(* IEC 61131-3 sources: ml2plc/examples/models/structured_text (part 8) *)

(* ---- test5_13k.st ---- *)
FUNCTION_BLOCK NeuralNetworkFB

VAR_INPUT
    input_data : ARRAY[0..4] OF REAL;
END_VAR

VAR_OUTPUT
    output_data : ARRAY[0..2] OF REAL;
END_VAR

VAR CONSTANT
    weights_0 : ARRAY[0..639] OF REAL := [0.087884, 0.019861, -0.120645, 0.107147, 0.108510, -0.209824, 0.028247, -0.067439, -0.017955, -0.147290, -0.044152, 0.074469, -0.058888, 0.021687, 0.118680, 0.075522, 0.073631, 0.110030, -0.236657, -0.068495, 0.032454, -0.131920, 0.026285, 0.065899, 0.005899, -0.086759, -0.068999, 0.126513, 0.120250, -0.038000, -0.006767, 0.065750, -0.029117, -0.015027, -0.120319, -0.212539, -0.105368, 0.074505, -0.034129, -0.051312, 0.169426, -0.112692, -0.026185, -0.089530, -0.065181, 0.010042, -0.051896, 0.010617, 0.083632, 0.159610, 0.026174, -0.171285, 0.004264, -0.070313, -0.094491, -0.141654, -0.152467, -0.156618, 0.092858, 0.118828, -0.052229, 0.008375, 0.033061, -0.192688, 0.001746, -0.046752, -0.129324, 0.150817, 0.004261, -0.119102, 0.039470, 0.110854, 0.036013, 0.111391, 0.032649, -0.101358, 0.029517, 0.081127, -0.131120, 0.030191, -0.073921, -0.066215, -0.138857, 0.117446, -0.204267, -0.076552, -0.113729, -0.110411, -0.046143, -0.050134, -0.177807, -0.017884, -0.068962, 0.016712, 0.066131, -0.097737, -0.106193, 0.097484, 0.054137, 0.121767, 0.109686, 0.092542, 0.089354, -0.074552, -0.203123, 0.140532, 0.141643, 0.060210, 0.020210, -0.161035, -0.144116, 0.140873, 0.103789, 0.073508, 0.004795, -0.115107, 0.086948, -0.059466, 0.117073, 0.013680, -0.031496, -0.164868, -0.113202, -0.082604, -0.006095, -0.168162, -0.110567, 0.046874, 0.136677, -0.073749, -0.155012, 0.014878, -0.081808, 0.120516, 0.058027, 0.145353, -0.058555, 0.169970, 0.055944, -0.106464, -0.128222, 0.048024, -0.034696, 0.045333, -0.081858, -0.044126, 0.116255, -0.032645, 0.032003, -0.076957, -0.143227, -0.022855, 0.031258, -0.128789, -0.003603, -0.048892, -0.177628, -0.061286, -0.205522, -0.115107, 0.037776, -0.058937, 0.105858, -0.171562, -0.111364, 0.005641, 0.013799, -0.030156, -0.012579, 0.138731, 0.152130, -0.132872, 0.006697, 0.030615, 0.032380, 0.099033, -0.036929, -0.106096, 0.088105, 0.045451, -0.001212, -0.054999, 0.011836, -0.200356, 0.118485, -0.131535, -0.076382, -0.113409, -0.136508, -0.098254, -0.114961, -0.107293, 0.082311, 0.142847, 0.215688, -0.091563, -0.096765, 0.206613, -0.199051, -0.171045, 0.031297, 0.036175, -0.169052, 0.002642, 0.031713, -0.080200, 0.119600, -0.076829, 0.080139, 0.087728, 0.077741, -0.114895, 0.089789, 0.080168, 0.076910, -0.097419, 0.053509, -0.025485, 0.138235, -0.007267, -0.163736, 0.012899, 0.039587, -0.003616, -0.071788, -0.133374, 0.202067, 0.095088, -0.135328, 0.047618, -0.138865, 0.097218, -0.084921, -0.171197, -0.132809, -0.030269, -0.199631, 0.071125, 0.096722, -0.117543, 0.109680, 0.125666, -0.187342, 0.017445, -0.181086, -0.113749, -0.160243, 0.146440, 0.145078, -0.233663, -0.124617, 0.020189, 0.104925, 0.091885, 0.136374, -0.015601, -0.137955, 0.067880, 0.188922, -0.114488, 0.006490, -0.073870, 0.020977, -0.157864, 0.083543, 0.024444, -0.012612, -0.184603, -0.155885, 0.037704, 0.041224, -0.191320, -0.026819, -0.137896, -0.026415, 0.037044, -0.009771, 0.196403, 0.007078, -0.052965, 0.021385, 0.019141, 0.128097, 0.099409, -0.082667, -0.044388, -0.141733, 0.008215, 0.058057, -0.006857, -0.162652, 0.131042, -0.070709, 0.116382, -0.018573, -0.097403, -0.185227, 0.072037, -0.193845, 0.027885, -0.064402, -0.099111, -0.093831, 0.008709, 0.068151, -0.170941, -0.121179, 0.017150, -0.059804, -0.133350, 0.123899, 0.176413, -0.016766, 0.089295, 0.127591, -0.040662, -0.062021, 0.035431, 0.069664, 0.023847, -0.041006, -0.117259, -0.124652, -0.044356, -0.079393, -0.063249, 0.124950, 0.164965, -0.199731, 0.063873, 0.134956, -0.238765, 0.055125, -0.055810, 0.051782, 0.056541, 0.108808, -0.073532, -0.077848, 0.123551, 0.024601, -0.120728, -0.004044, 0.112966, -0.161989, 0.012075, -0.070966, -0.124047, 0.167929, 0.125195, 0.098143, -0.096104, 0.166867, 0.114795, -0.136621, -0.019339, 0.168998, -0.007273, 0.138194, 0.038277, 0.112113, -0.097517, 0.167485, 0.052191, -0.080308, 0.085419, 0.078983, -0.111131, -0.060336, -0.188764, 0.007864, 0.047479, -0.094697, 0.132104, -0.231222, -0.136076, 0.007164, 0.140243, 0.200802, -0.160538, 0.028893, 0.105251, -0.087435, -0.023133, -0.181240, 0.031476, -0.069354, 0.025107, 0.003484, 0.017893, 0.013283, 0.086928, 0.116381, -0.105047, -0.011669, -0.144326, -0.081993, 0.015335, 0.162402, 0.170721, -0.073380, -0.064310, 0.021418, -0.052916, -0.194195, -0.104925, 0.077744, -0.046308, 0.041450, 0.123528, -0.009889, 0.048534, -0.204614, 0.114375, -0.007900, -0.096067, -0.144443, 0.066950, -0.017162, 0.127650, -0.021940, -0.186933, -0.174070, 0.114869, 0.013821, 0.049158, 0.118836, 0.110080, -0.179380, -0.145327, -0.151734, -0.067201, 0.090523, -0.180013, -0.111317, 0.028459, 0.011573, 0.167342, 0.032929, -0.037529, 0.162289, 0.121033, 0.033484, 0.080197, -0.115669, -0.150395, 0.122810, -0.140164, 0.012817, -0.085399, -0.030360, 0.052412, 0.199205, -0.085308, 0.099355, -0.185208, -0.119913, 0.022915, -0.003856, 0.096522, -0.164929, -0.085813, -0.083492, 0.066105, -0.127158, 0.160928, 0.150646, -0.064350, -0.094705, 0.068810, 0.104658, 0.100290, 0.016024, 0.107678, 0.176333, 0.074564, -0.097281, -0.158018, -0.189581, -0.098518, -0.040255, -0.200370, -0.032509, -0.113215, -0.046972, -0.175030, 0.121636, 0.006522, 0.068477, 0.060772, -0.172631, 0.022521, -0.104405, -0.176789, 0.053084, -0.234425, -0.225009, 0.077532, 0.060609, -0.072898, -0.043883, -0.159845, 0.054400, -0.060357, 0.152364, 0.075698, -0.101363, 0.156116, -0.068740, -0.008421, 0.115683, -0.032726, 0.049882, 0.060400, -0.041212, -0.130228, 0.171733, -0.081668, -0.138404, 0.156815, -0.057446, 0.156922, 0.138291, 0.004256, 0.156900, -0.256590, -0.045184, 0.056040, 0.093967, -0.093704, 0.088963, -0.071382, 0.138222, 0.082414, 0.019420, 0.140588, -0.114552, -0.081097, -0.043554, -0.027499, -0.167955, 0.141868, 0.030455, 0.116915, 0.078890, -0.036069, -0.054053, 0.126143, 0.016059, 0.096736, 0.161875, 0.148323, -0.004357, -0.166265, -0.138691, 0.038991, 0.137727, 0.012094, -0.163153, -0.058560, -0.009588, -0.142637, -0.131980, 0.059672, -0.001274, -0.182290, -0.218865, -0.117359, -0.147914, 0.161844, -0.171897, -0.093763, 0.165442, 0.016261, -0.184435, -0.071222, 0.075867, -0.019360, -0.157325, -0.025250, -0.191039, 0.152266, -0.070228, -0.082297, 0.103244, -0.262244, 0.154374, 0.147566, -0.188977, -0.058970, 0.071598, 0.084986, -0.117181, -0.221621, -0.140587, -0.165058, 0.133049, -0.004266, -0.108147, 0.034074, -0.004569, -0.023090, 0.005967, -0.013832, -0.056172, 0.101765, -0.228049, 0.212225, -0.149336, -0.038122, -0.155115, 0.051004, -0.012800, 0.093140, -0.253202, -0.082567, -0.049787, 0.180747, -0.041803, 0.003407, 0.064646, 0.024799, -0.096398, 0.025533, -0.177775, -0.043537, -0.056790, -0.013036, -0.173823, 0.109881, 0.120896, 0.023794, -0.107422, -0.086024, 0.180928, -0.020671, 0.083740, 0.123611, 0.087525, 0.156801];
    bias_0 : ARRAY[0..127] OF REAL := [-0.138056, -0.724342, -0.149341, -0.281606, -0.725367, 0.232611, -0.248216, -0.224301, -0.455382, -0.588808, 0.331585, -0.105728, -0.004159, 0.141275, -0.052369, -0.498210, -0.228472, 0.128578, -0.324100, -0.114577, -0.552493, -0.092725, -0.231976, -0.594564, 1.152468, 0.320418, 1.080323, -0.436585, -0.201718, -0.644658, -0.083568, 0.892163, -0.533870, 0.395853, 0.012269, 0.399186, -0.090490, -0.443884, 0.422784, 0.699066, 0.525596, -0.248559, 0.707993, 0.283335, 0.051301, 0.005778, 0.071785, 0.709974, -0.306237, 0.124496, 0.201839, -0.570137, -0.169047, -0.182123, 0.495954, -0.100448, 1.026744, -0.484968, 0.789213, 0.337440, 0.164353, -0.134713, -0.277190, 0.014476, -0.957523, -0.088268, 0.004471, -0.558361, 0.308556, -0.375165, -0.692890, 0.276062, 0.256898, 0.133769, -0.481402, -0.289402, -0.027431, 0.037170, 0.774907, -0.558535, -0.040130, 0.377911, 0.574793, 0.486151, 0.168924, 0.406046, 0.144867, -0.593385, 0.075902, -0.426114, -0.372866, 0.453651, -0.236809, -0.562530, 0.037890, -0.083074, -0.047217, 0.078249, 0.167289, -0.330759, -0.283430, -0.460562, -0.174557, 0.892016, -0.115629, -0.579056, 0.747610, -0.564211, -0.082146, 0.059292, 0.430699, 0.005029, 0.198333, -0.513879, 0.096918, 0.126206, 0.071723, -0.133315, -0.245988, 0.964687, -0.703479, 0.089156, -0.414976, -0.108005, -0.900232, -0.744488, -0.873102, -0.797852];

    weights_1 : ARRAY[0..12287] OF REAL := [-0.081575, -0.080771, 0.015952, -0.039088, -0.116122, 0.043837, 0.081503, -0.146702, -0.097420, 0.123321, -0.143534, 0.087642, -0.013072, 0.120403, -0.032723, -0.019567, 0.109142, 0.046921, -0.151230, 0.034047, 0.068958, -0.110997, -0.006236, 0.099731, 0.103434, -0.019739, 0.061900, -0.030395, -0.006606, 0.042065, 0.125518, -0.158020, -0.060671, -0.011133, -0.174419, -0.000909, -0.087395, 0.107763, 0.032645, -0.159583, 0.019297, -0.055804, 0.041226, -0.102607, 0.111457, 0.036441, 0.020504, 0.026678, 0.022357, 0.058828, 0.009128, -0.137546, 0.099089, -0.132678, -0.139020, -0.078414, 0.134850, -0.109238, -0.088241, 0.086606, -0.129975, -0.106856, -0.173047, 0.002129, 0.073779, -0.001719, 0.012466, -0.149798, 0.068260, 0.018230, -0.073247, 0.025459, -0.025935, -0.083550, -0.014844, 0.044535, 0.024790, 0.031258, 0.047537, -0.126853, 0.030907, -0.174494, 0.123196, -0.139801, -0.101418, -0.042713, -0.031737, -0.139095, -0.141767, 0.051548, -0.103749, -0.134006, 0.124273, 0.033699, 0.088179, -0.196681, -0.061558, -0.097976, 0.041162, -0.066488, -0.223767, -0.156958, 0.119515, 0.030284, 0.064781, 0.065118, -0.019679, -0.014793, 0.070956, 0.005814, -0.125978, 0.148016, -0.176253, -0.110496, -0.086278, -0.064303, 0.029931, 0.013686, 0.164138, -0.022327, -0.030191, 0.187196, -0.098539, -0.023848, 0.048127, -0.111411, -0.095664, -0.256552, 0.008552, -0.103314, 0.051327, -0.022576, -0.091046, 0.019166, -0.099166, -0.173986, -0.026153, 0.027388, -0.109343, 0.046421, 0.037128, -0.124205, -0.198771, 0.073731, -0.039520, 0.016815, -0.047930, -0.129724, 0.019335, -0.119635, -0.026225, -0.029072, 0.158678, -0.173663, 0.027847, -0.049243, -0.020055, -0.109040, 0.095462, -0.042686, 0.151513, -0.077091, -0.131769, 0.054254, 0.026624, -0.155398, -0.082870, -0.159275, 0.059890, 0.062534, -0.142575, -0.059085, -0.185808, -0.137954, -0.029401, 0.077038, 0.112156, 0.029459, 0.065796, 0.013224, -0.179952, -0.117919, -0.115410, 0.092213, 0.008067, 0.144769, -0.132419, 0.141382, -0.085988, -0.073259, -0.108810, -0.089521, 0.090714, 0.070094, 0.051771, -0.198376, 0.097630, 0.134390, 0.070879, -0.084352, -0.077932, -0.084724, 0.013531, 0.103697, 0.083068, -0.022807, -0.099833, 0.026875, -0.011101, 0.100574, -0.189504, 0.008358, -0.130581, -0.017598, 0.049774, -0.038556, -0.034455, 0.092771, 0.008732, -0.099842, -0.203902, 0.097001, 0.054298, 0.068758, -0.017547, -0.119806, -0.001483, 0.150792, 0.059175, -0.024380, 0.077527, -0.089932, -0.095934, 0.067083, 0.051638, -0.140169, 0.016767, -0.031886, -0.077586, -0.156478, 0.136940, -0.068401, -0.156731, -0.031153, 0.027569, -0.069691, 0.016632, 0.085590, -0.087230, -0.124976, 0.178376, 0.054593, 0.139863, 0.138583, -0.028121, -0.011154, -0.060567, -0.100126, -0.094427, -0.078613, -0.021682, -0.123174, -0.107229, 0.095945, -0.081012, -0.122688, -0.075887, -0.142662, -0.036621, -0.064916, -0.071555, 0.096564, 0.021082, 0.004940, 0.073835, 0.102978, 0.013753, -0.087000, -0.023456, -0.025726, 0.041069, 0.019725, -0.170109, -0.065330, -0.065098, -0.043905, -0.013389, -0.033329, 0.077615, 0.045581, -0.113043, -0.026083, -0.092637, 0.131571, 0.111947, 0.053334, 0.064196, -0.046716, -0.096859, -0.185973, -0.034940, 0.044770, -0.124819, 0.029667, -0.082584, -0.149761, -0.067224, 0.100945, 0.101797, -0.123318, 0.079437, -0.170388, 0.043855, -0.096770, 0.093361, -0.037078, -0.054357, -0.136876, 0.030271, 0.088059, -0.158535, 0.016276, -0.199991, -0.136451, -0.101051, -0.099338, -0.051318, -0.091107, -0.092926, 0.125917, 0.120004, 0.099235, 0.054448, -0.054184, -0.088516, 0.031720, -0.110417, 0.021548, 0.114272, 0.104105, -0.029168, -0.104910, 0.043389, 0.110131, 0.067098, 0.063883, 0.125061, -0.140973, -0.087429, -0.183545, 0.001501, 0.090085, 0.090463, -0.068449, 0.104290, -0.047815, -0.107690, 0.142746, -0.009204, -0.074146, 0.109043, -0.056259, 0.005365, -0.095835, -0.019732, -0.090880, -0.179324, -0.144838, 0.008955, -0.031656, -0.153258, -0.049975, -0.136535, -0.153729, -0.007882, 0.076208, -0.147986, 0.120409, -0.050599, 0.102071, 0.002109, -0.156943, -0.029278, -0.102693, -0.051444, 0.111964, 0.059902, -0.168826, -0.068986, -0.174917, 0.080254, 0.004751, 0.066618, 0.096905, 0.066631, -0.175463, 0.091283, -0.263883, 0.056194, 0.079930, -0.117990, -0.009883, 0.138474, -0.146369, -0.138613, -0.192223, -0.044161, 0.087972, 0.023354, 0.044543, 0.110326, -0.011888, 0.100713, 0.032271, -0.142762, -0.173276, -0.082045, -0.071345, -0.156709, -0.059416, 0.024078, 0.016129, 0.006350, -0.202165, -0.177114, 0.204796, 0.039982, -0.145523, 0.047530, -0.165438, 0.029745, -0.033077, 0.192667, -0.125515, -0.130639, 0.063787, -0.023226, 0.007809, -0.015500, 0.005910, 0.012534, -0.158731, -0.177921, -0.028937, -0.156686, -0.188195, 0.135282, 0.209456, 0.003387, -0.116251, -0.139349, 0.030706, 0.084070, 0.139131, -0.130020, 0.098266, -0.017343, -0.102753, -0.081793, -0.108168, 0.015434, -0.063223, -0.088817, 0.008182, 0.044385, 0.194167, 0.068721, 0.144784, -0.144739, 0.149692, -0.122958, 0.034189, -0.118378, -0.035300, -0.031611, -0.090980, 0.098072, -0.082291, 0.040535, 0.028408, 0.077057, 0.016835, -0.177612, -0.111623, 0.112017, -0.175378, 0.122941, 0.071300, -0.029213, -0.042673, -0.095251, 0.091868, -0.124875, 0.123380, 0.094310, -0.056404, 0.101097, -0.187158, -0.099725, -0.074531, -0.119461, -0.089910, 0.027321, -0.089037, -0.095327, -0.095788, 0.158980, -0.080355, 0.051269, -0.036277, 0.013874, 0.087641, 0.023480, -0.123195, -0.114087, 0.079653, -0.005070, 0.083194, 0.071204, -0.012910, -0.128791, -0.214303, 0.041115, -0.126938, 0.010794, -0.104911, -0.167860, -0.056907, 0.149767, 0.072014, 0.018457, -0.003708, -0.084242, 0.034660, 0.148553, 0.060466, 0.050078, 0.173174, -0.156669, 0.012732, -0.156297, -0.083725, -0.087539, -0.276414, -0.029359, -0.057753, 0.001603, 0.126020, -0.011550, 0.082022, -0.048681, -0.161668, 0.021370, 0.141360, -0.130907, -0.191119, -0.010477, -0.036678, -0.091980, 0.101416, -0.012654, -0.061183, -0.145007, 0.024690, 0.037292, 0.001704, 0.096528, -0.209641, 0.002475, -0.044156, -0.063900, 0.157965, -0.209313, 0.107978, -0.030685, 0.127991, 0.088548, -0.137926, -0.008005, -0.103959, 0.038476, 0.099615, -0.041820, 0.010803, -0.100065, 0.066539, -0.149380, 0.131097, -0.141308, -0.049057, -0.054971, -0.036114, 0.115146, -0.148750, -0.126427, -0.078635, -0.048640, -0.046237, -0.130117, 0.004752, 0.102776, -0.069640, 0.024115, -0.109310, -0.096013, 0.116772, -0.136342, -0.151241, -0.199084, 0.039571, 0.116098, -0.054730, -0.043315, 0.050230, 0.093377, -0.058800, 0.043897, -0.096458, 0.167670, -0.171068, 0.003364, -0.012613, 0.132328, 0.043677, 0.004500, -0.052957, -0.181461, 0.092122, 0.161901, -0.018877, 0.097804, -0.101418, 0.057685, 0.046452, 0.063500, -0.149884, -0.077202, -0.050282, 0.062265, -0.133137, 0.094386, -0.027847, 0.003860, -0.058797, 0.096755, 0.133752, 0.018234, 0.115755, -0.137680, 0.030889, -0.043614, 0.082428, 0.045449, 0.049964, 0.031676, -0.006952, -0.006175, -0.060989, 0.016020, -0.001273, -0.129249, -0.027272, -0.145721, 0.129620, 0.032681, -0.020259, 0.089839, -0.076454, 0.031277, -0.137930, -0.190245, -0.092762, -0.169273, -0.125275, 0.042772, -0.150519, -0.108547, -0.041230, -0.111160, -0.003413, -0.131887, 0.051243, -0.094373, 0.115747, 0.035868, -0.115496, -0.008602, -0.121400, -0.088105, 0.047530, 0.094965, -0.057794, 0.045937, 0.047745, -0.151089, 0.135993, 0.068231, -0.079802, -0.143148, -0.122689, 0.037814, -0.170841, 0.047921, -0.078489, -0.068901, -0.145030, -0.124568, 0.037971, -0.112618, 0.090066, 0.053041, -0.113300, 0.042961, 0.100212, -0.056396, -0.114706, -0.163505, -0.130223, -0.165611, -0.038295, 0.013722, -0.089551, -0.117751, -0.038264, 0.169660, -0.045797, -0.036698, -0.141689, -0.065967, -0.000077, 0.019098, -0.069963, -0.092839, -0.101812, -0.004868, -0.023554, -0.133523, -0.142896, 0.034829, 0.025655, 0.172733, -0.116783, 0.116567, 0.077891, 0.170584, 0.107316, -0.126802, -0.021477, -0.087033, 0.107559, -0.062535, 0.110244, -0.020078, 0.006528, -0.196714, -0.008804, -0.034624, -0.037185, -0.040095, -0.127234, -0.015266, -0.029318, 0.098768, 0.070560, -0.188236, 0.091512, 0.072778, -0.121254, -0.142115, -0.102058, -0.126129, -0.144473, 0.047309, 0.031633, 0.111848, 0.022209, 0.000316, -0.103872, -0.152406, 0.063265, -0.086201, -0.049895, -0.128511, -0.042608, -0.013025, 0.129606, -0.152738, 0.091822, -0.170736, -0.122971, 0.036491, -0.103669, -0.093657, 0.065951, 0.086443, -0.007772, 0.126724, 0.061812, 0.073030, -0.227505, -0.150730, -0.152455, 0.003632, -0.019424, -0.054101, 0.081972, 0.112612, 0.019746, 0.076702, 0.212985, -0.150149, -0.038424, -0.126008, 0.020174, -0.003787, -0.029846, 0.013167, 0.071178, -0.081888, 0.097691, 0.020292, 0.018873, -0.140535, 0.051663, -0.155505, 0.038109, -0.005970, 0.018861, 0.061807, 0.091283, 0.099963, 0.122483, 0.048785, 0.033977, 0.041410, 0.140400, -0.092338, 0.112759, 0.076005, -0.133343, -0.162613, -0.008164, -0.002846, 0.120728, -0.049317, 0.054437, -0.127069, 0.042041, -0.035214, 0.139597, 0.073649, -0.101931, -0.016045, 0.181245, -0.043369, 0.026610, -0.137698, 0.167959, 0.122667, -0.008332, 0.021051, 0.040108, -0.156969, -0.068006, 0.137933, 0.012884, -0.106799, -0.009552, -0.219680, -0.027378, 0.057219, -0.206282, 0.012929, -0.139442, 0.068162, -0.159516, 0.096407, -0.083495, -0.205347, 0.011081, 0.048977, -0.011546, 0.089416, -0.219959, -0.146311, 0.047244, 0.006085, 0.036988, 0.133529, 0.083324, -0.074794, -0.099529, -0.002222, -0.047307, -0.030684, -0.177784, -0.093368, -0.141561, 0.078858, 0.135456, -0.166646, 0.034251, -0.020081, 0.068057, -0.141532, 0.075862, 0.065621, -0.052889, -0.186487, 0.010214, -0.061436, -0.028441, 0.125152, -0.036969, 0.058498, 0.044020, 0.165813, -0.125980, -0.033366, -0.174131, -0.125943, 0.055094, -0.088112, 0.035833, 0.041747, 0.076717, 0.076765, -0.016334, -0.119987, -0.135628, 0.015400, 0.005722, 0.006286, -0.129062, -0.029350, -0.044798, 0.037943, 0.126117, -0.132406, 0.036613, -0.112067, -0.031121, 0.100631, -0.012509, 0.072480, 0.034916, -0.040505, 0.007290, 0.049140, 0.149019, -0.092554, -0.042404, 0.068616, 0.132734, 0.003138, 0.170876, -0.031358, -0.155839, -0.081269, 0.042707, -0.034900, 0.220723, -0.018079, 0.113232, -0.039536, -0.035911, 0.146646, 0.089903, 0.006342, -0.012555, 0.067873, -0.115261, 0.082812, 0.164852, 0.084914, 0.086952, -0.101140, 0.065694, 0.004201, 0.021580, -0.042629, 0.105508, -0.085644, 0.183658, 0.178939, 0.059744, -0.124989, -0.095250, -0.118859, 0.001045, -0.026453, 0.015741, -0.001020, -0.147134, 0.057491, 0.033330, 0.098456, 0.085774, -0.069800, 0.053079, 0.116645, 0.082423, -0.088994, 0.040234, -0.084737, -0.119974, -0.002935, -0.071704, 0.159501, 0.157314, -0.116031, -0.094580, 0.004709, -0.090457, 0.034409, -0.098700, -0.012167, 0.037498, -0.034314, 0.049258, 0.043418, -0.047919, -0.128354, -0.004897, -0.122908, 0.149899, 0.089695, 0.137241, -0.001262, 0.026590, 0.062069, -0.022439, 0.013561, 0.108820, -0.134295, 0.137737, -0.104128, 0.029637, 0.102498, 0.075547, 0.098281, 0.107930, -0.099356, -0.012938, -0.020183, -0.223851, 0.043924, 0.107465, 0.156199, -0.088132, 0.188467, 0.102066, 0.064692, -0.090133, -0.001347, -0.082854, 0.183009, -0.038977, -0.159207, 0.057301, -0.136873, 0.048873, 0.031771, -0.171822, 0.033120, 0.105704, -0.084895, 0.095055, 0.137444, -0.163820, 0.112387, 0.051031, -0.072802, -0.100967, 0.013958, 0.075336, -0.143393, -0.055055, -0.117185, 0.108107, 0.162765, -0.049701, -0.010500, -0.129675, 0.059109, -0.169230, 0.061079, -0.012083, -0.151733, 0.007924, -0.064643, -0.044676, -0.096629, -0.106404, 0.128860, -0.123374, 0.097159, 0.044151, -0.102661, -0.142225, -0.094126, -0.005144, -0.182815, 0.042802, -0.011589, -0.081280, -0.168038, 0.082915, -0.112574, -0.051578, -0.001187, -0.026704, -0.091962, -0.026611, -0.171998, -0.021113, 0.140911, -0.098982, 0.098242, 0.080007, 0.037016, -0.078325, 0.135061, 0.078783, -0.140612, 0.098578, -0.096234, 0.081160, -0.122356, -0.113938, -0.164598, 0.011331, -0.139634, -0.015426, 0.157431, -0.172702, 0.099078, -0.018352, 0.028085, -0.102126, 0.009692, -0.057786, -0.068308, 0.046532, 0.022939, 0.047090, 0.057643, 0.101340, 0.031700, -0.155278, 0.025313, -0.162245, 0.062350, 0.080738, 0.009415, -0.026625, 0.119341, -0.115887, 0.043791, 0.043181, 0.113826, -0.121817, 0.102165, -0.069487, 0.006380, 0.074927, 0.043731, 0.147266, 0.039980, -0.006088, -0.082346, -0.193183, -0.022871, -0.117219, 0.016636, -0.028051, -0.106046, -0.005760, 0.153666, -0.068575, 0.080032, 0.041547, -0.070853, -0.039723, -0.133037, 0.124683, -0.105086, -0.130024, -0.122982, -0.097882, -0.166385, 0.096523, -0.060713, 0.046434, -0.158093, 0.057526, 0.090288, 0.091276, 0.087174, -0.018942, -0.022930, 0.028879, 0.081154, 0.050385, -0.228233, 0.075629, -0.141450, 0.016981, -0.003183, -0.011411, -0.034834, 0.062535, -0.140759, -0.069517, -0.054256, -0.126463, 0.062169, -0.071767, 0.063638, 0.035320, 0.025509, -0.102183, -0.013740, -0.105443, 0.067947, -0.093319, 0.066332, 0.001127, -0.230074, -0.032940, -0.024680, -0.075319, 0.104570, -0.063355, 0.042160, -0.083321, 0.096235, -0.054556, 0.046468, -0.142220, -0.152431, -0.080084, -0.034122, -0.039364, 0.021040, -0.121876, -0.047387, -0.016643, -0.075452, 0.011071, -0.096630, 0.167191, -0.022463, -0.161584, -0.114355, -0.013775, -0.212787, 0.114291, 0.148954, -0.270307, -0.044340, -0.038644, -0.130380, 0.008371, 0.179310, 0.028057, -0.112501, 0.099296, -0.023552, 0.042440, -0.223643, -0.089552, 0.121801, -0.101898, 0.101719, -0.019475, -0.138102, 0.007500, 0.114520, -0.020841, 0.078318, -0.146791, -0.159486, -0.033819, -0.108025, 0.019645, -0.240050, -0.094725, 0.001863, -0.061960, 0.070538, 0.037391, -0.004894, -0.129432, -0.039346, -0.016018, 0.048675, 0.183405, -0.061341, 0.044579, -0.075781, -0.090313, -0.061431, -0.242545, 0.149409, 0.192036, 0.042303, -0.174307, -0.174971, 0.118598, -0.012059, 0.008028, -0.051703, 0.072126, 0.039219, -0.051813, -0.157609, -0.053761, 0.077431, -0.167700, -0.136599, -0.126247, -0.083612, 0.061878, -0.069953, 0.017028, -0.059142, -0.105931, 0.065761, -0.230763, 0.098776, -0.233016, 0.107031, -0.091945, -0.140657, 0.106068, -0.168658, 0.117609, -0.162881, -0.062493, -0.031648, -0.215897, -0.011096, -0.223865, -0.194450, 0.018461, -0.098600, 0.019417, -0.010198, 0.121387, -0.085882, 0.033285, 0.064565, -0.101164, -0.154355, -0.008463, -0.022031, 0.086821, 0.073677, -0.047492, -0.006241, -0.083720, -0.064338, -0.030201, 0.068820, -0.012762, 0.006955, -0.069824, 0.048148, -0.098935, -0.074085, -0.131027, -0.048977, -0.079691, 0.061712, -0.017702, 0.047844, -0.149083, -0.174584, -0.017555, -0.069080, 0.057426, 0.023185, 0.094438, 0.055650, -0.178939, 0.114310, -0.196780, -0.032571, -0.060820, -0.076543, 0.022690, 0.098297, -0.095817, 0.016638, 0.011793, -0.101782, 0.005777, -0.149359, 0.027835, -0.077289, 0.092431, -0.093891, 0.010222, 0.012915, -0.102511, -0.031433, -0.139489, -0.131653, -0.133860, -0.170684, 0.000861, 0.176236, 0.023889, -0.122425, 0.031023, -0.042648, -0.200706, -0.007618, -0.172353, -0.060969, -0.111408, 0.035170, 0.026013, -0.059565, 0.163137, 0.100273, 0.142385, 0.054498, -0.210962, 0.083249, -0.172852, 0.049680, 0.061989, 0.080453, 0.054906, 0.060045, -0.137977, -0.005662, 0.011224, 0.083500, 0.057573, -0.103310, 0.014571, 0.012037, -0.127015, -0.040393, -0.106786, -0.132445, -0.089465, 0.053720, -0.111644, -0.152595, -0.072208, -0.170288, 0.040783, -0.051353, -0.123556, -0.059620, -0.006337, 0.053879, 0.018863, 0.178810, -0.048635, 0.011481, 0.031570, 0.134769, -0.086727, 0.057939, -0.112196, -0.124786, -0.037214, -0.183068, 0.051824, 0.088464, 0.170947, -0.089516, -0.101557, -0.023134, 0.039533, -0.137372, -0.068921, 0.120034, -0.064358, -0.211081, 0.050003, 0.097631, -0.164230, -0.003052, -0.045674, 0.033500, -0.155961, 0.149210, -0.005820, -0.095616, -0.008706, -0.073449, -0.007479, -0.065913, 0.011839, 0.061956, -0.159078, -0.007190, 0.028311, -0.068458, -0.032719, -0.096845, 0.000351, 0.083672, -0.176350, -0.101202, -0.156637, 0.120088, -0.090894, 0.074344, -0.097555, -0.069346, -0.097220, 0.005215, -0.199269, -0.075000, -0.012239, -0.153847, -0.132105, -0.173554, -0.022580, -0.075864, 0.072241, -0.179801, 0.114656, 0.058945, 0.032403, -0.035467, -0.073135, -0.026923, -0.004199, 0.126423, -0.123071, 0.024513, 0.119495, -0.079067, 0.107798, -0.002691, -0.177214, -0.080168, 0.087260, 0.083324, -0.036822, 0.012710, 0.006805, 0.025345, 0.014063, 0.139339, 0.068182, -0.163975, -0.018243, -0.111255, 0.011790, 0.047546, 0.092633, 0.049318, 0.003007, -0.145426, 0.051505, 0.019591, 0.038348, 0.106809, 0.146770, -0.137394, 0.023419, -0.104374, 0.015242, -0.077740, -0.014287, 0.107080, 0.149179, -0.032868, 0.014391, 0.112384, -0.140490, 0.000523, 0.038513, 0.085826, 0.033327, 0.122935, 0.068390, 0.046117, 0.030794, -0.186023, -0.078125, -0.018852, 0.109274, 0.066455, 0.017141, -0.133333, -0.193708, -0.146445, -0.015501, 0.026529, 0.082395, 0.149612, -0.070591, -0.016908, -0.059412, 0.034737, -0.125785, -0.132630, 0.051595, -0.068432, 0.058917, -0.063994, -0.020062, -0.155251, -0.130603, -0.102926, -0.068344, 0.223298, 0.114052, 0.093608, -0.056596, 0.014436, 0.056514, 0.053748, 0.041788, -0.013315, -0.054554, -0.021707, -0.017912, -0.076426, -0.065880, -0.060482, 0.059109, 0.033523, -0.065950, 0.130728, 0.155523, -0.122129, 0.097537, -0.222720, -0.033999, -0.179547, 0.132113, -0.132758, -0.163402, -0.097568, 0.081810, -0.063774, -0.237891, -0.098302, 0.001285, -0.002167, -0.148563, -0.078971, -0.102606, -0.169557, -0.090034, 0.104811, 0.052321, 0.137128, 0.028810, -0.102812, 0.046596, 0.095611, -0.091704, -0.122140, -0.040893, 0.128003, -0.118820, 0.079260, -0.053132, 0.120491, 0.065923, 0.101679, -0.118584, -0.076018, 0.031019, -0.158750, 0.066865, 0.156857, 0.124133, 0.072551, 0.136147, -0.068172, -0.190488, -0.019130, 0.084109, -0.069187, 0.136179, -0.005778, 0.083175, 0.004151, -0.108535, 0.124859, -0.054482, -0.019212, -0.051216, 0.151764, -0.133774, 0.026327, -0.140163, -0.237679, -0.014108, 0.064628, 0.025393, -0.200114, -0.067511, -0.001822, -0.160585, -0.037121, -0.149930, 0.102790, -0.021203, -0.122963, -0.091361, 0.006626, -0.123720, 0.008464, 0.025206, -0.143426, 0.050645, -0.066107, -0.114658, 0.021127, -0.077297, 0.020617, -0.055209, -0.196839, 0.019999, -0.047371, 0.108169, -0.014506, -0.082857, 0.090321, -0.072653, 0.029153, -0.007638, 0.054287, -0.066536, 0.103992, -0.068357, 0.043941, -0.139107, -0.132066, 0.079844, 0.038007, -0.042187, -0.056770, 0.086439, 0.099471, 0.056606, -0.120636, 0.073782, 0.127915, -0.159352, 0.139489, -0.109178, -0.001992, -0.091596, -0.132664, -0.016212, 0.041536, 0.108049, 0.085386, 0.068069, -0.030001, -0.029575, -0.137504, 0.113700, 0.117755, 0.133271, -0.015861, -0.094789, -0.130660, -0.131559, -0.135082, -0.177463, -0.057344, 0.001805, 0.136894, -0.146070, -0.103945, -0.151248, 0.062254, -0.020492, -0.017738, 0.082921, 0.042381, -0.109089, -0.128478, 0.002673, -0.000820, 0.111654, 0.098417, 0.104491, -0.044083, 0.144458, 0.042958, -0.115993, -0.112584, -0.192943, 0.022451, 0.017492, -0.054143, 0.040774, 0.133315, -0.069498, -0.079107, -0.064530, 0.116959, 0.105073, -0.058618, 0.066981, 0.110520, -0.144423, 0.052642, 0.093975, -0.149870, -0.052229, -0.001838, 0.011842, -0.085902, 0.147386, -0.059832, -0.049631, -0.042176, -0.175652, -0.072840, -0.031563, -0.112192, 0.084438, -0.114146, -0.094277, -0.112050, 0.000733, -0.171038, -0.045380, -0.079449, 0.126015, -0.108049, -0.208123, -0.046716, -0.193074, -0.061850, -0.156245, 0.102635, 0.133027, 0.053019, 0.095702, -0.069115, 0.134063, 0.129244, -0.039284, 0.024840, -0.002832, 0.003597, -0.088943, 0.082234, 0.073630, 0.102140, -0.006331, 0.014311, 0.078271, -0.088671, 0.122475, -0.099081, -0.042141, 0.071669, 0.087143, 0.093409, 0.028684, -0.099658, -0.022964, -0.073099, 0.074543, -0.151403, 0.114005, 0.093944, -0.021708, 0.104447, -0.085412, 0.053264, 0.121513, -0.109735, -0.168127, 0.097666, 0.119226, -0.030115, -0.049430, 0.060198, -0.012868, -0.016367, -0.138113, -0.145767, -0.009954, 0.013421, -0.126789, 0.056323, 0.116540, 0.010144, 0.100273, -0.079003, 0.124674, 0.142510, 0.035960, -0.160469, -0.118609, -0.177625, -0.066986, 0.061048, -0.183329, -0.144361, -0.094739, -0.051829, -0.079642, -0.107499, -0.153177, 0.129971, -0.110818, 0.028459, -0.109879, 0.093607, -0.010001, -0.146904, -0.124400, 0.069906, -0.151181, -0.136660, -0.132783, -0.029697, -0.035066, 0.066000, -0.000677, 0.103650, -0.037971, 0.019022, -0.057398, -0.089334, -0.149536, 0.098794, 0.086038, 0.018742, -0.149346, -0.059685, 0.100798, -0.072522, -0.016912, -0.024436, -0.013465, 0.146220, 0.026841, 0.122860, -0.184557, -0.000641, -0.171788, 0.037912, -0.007957, -0.029495, 0.072551, 0.019778, -0.033822, 0.017165, -0.074381, -0.010408, -0.108626, -0.107838, -0.161565, -0.167354, 0.053410, 0.083216, 0.061002, 0.002115, 0.069332, 0.127145, -0.065106, -0.074354, -0.123912, 0.031066, 0.006686, -0.089992, -0.149129, -0.119466, -0.104320, 0.050860, -0.143835, 0.147742, -0.002157, 0.074529, 0.178429, -0.044086, -0.104907, -0.089663, -0.042856, 0.104700, -0.088354, 0.031053, -0.100033, -0.032134, 0.149250, -0.038932, -0.014376, -0.021739, -0.093341, -0.054363, 0.108898, 0.114017, -0.086645, 0.083144, 0.090645, 0.098105, -0.022636, -0.052745, -0.018285, -0.041028, 0.034169, -0.079790, 0.115126, -0.123778, -0.065468, -0.003593, -0.107618, -0.035261, 0.040267, 0.132502, -0.022881, -0.037396, 0.036865, 0.099346, 0.039147, 0.115031, 0.120937, 0.047241, -0.046646, -0.107199, -0.020799, 0.046719, 0.079567, -0.011353, -0.114912, -0.075716, 0.116529, 0.170175, -0.155336, 0.015451, 0.102393, 0.019118, 0.028938, -0.028650, 0.025321, -0.027877, 0.133061, -0.088561, 0.060552, -0.029265, 0.070461, 0.073477, -0.011742, -0.051259, -0.009950, -0.211257, -0.146422, -0.049485, -0.006472, 0.124575, 0.073940, 0.081784, -0.108216, 0.011725, 0.003865, 0.044620, 0.113047, 0.038560, -0.182095, 0.020173, 0.058980, -0.120819, 0.071411, 0.085430, -0.070545, -0.028030, 0.113139, 0.092983, 0.042718, 0.113072, 0.139558, -0.043894, -0.152012, -0.104219, 0.025752, -0.147279, 0.084490, 0.106674, 0.068585, 0.071614, -0.142347, 0.002176, 0.214158, -0.113199, 0.046227, 0.128078, 0.039199, 0.010803, 0.072642, -0.089259, 0.078605, 0.018934, -0.102213, -0.063443, 0.032506, 0.147601, 0.015410, -0.148183, -0.070211, -0.081848, 0.077835, -0.123323, -0.061873, -0.007263, 0.110577, 0.030356, 0.002538, 0.169235, 0.089196, -0.053361, -0.089864, -0.090295, 0.060608, -0.099190, -0.031970, -0.025033, 0.086945, 0.154570, -0.039876, -0.180524, -0.168219, 0.045183, -0.052669, -0.083731, 0.029555, -0.084492, -0.004269, -0.078340, -0.053816, -0.140037, -0.132298, -0.063039, -0.095315, 0.075391, 0.048750, 0.144273, 0.123816, 0.118897, -0.159599, 0.061557, 0.056293, 0.092460, -0.166436, -0.044038, 0.023204, -0.049447, -0.075780, 0.080488, 0.034385, -0.053538, 0.031551, 0.144702, -0.140288, 0.020236, -0.099793, -0.133896, 0.013519, -0.083978, -0.188188, -0.166063, -0.084991, 0.002957, -0.081795, -0.060523, -0.128160, -0.038911, 0.000799, -0.030651, -0.142306, -0.002057, -0.121196, -0.079845, 0.007848, -0.131672, 0.138943, -0.157043, -0.106167, -0.148926, -0.144106, -0.076408, 0.155239, -0.042559, -0.091393, -0.179282, 0.062463, -0.187367, -0.016946, 0.000128, 0.036851, -0.176733, -0.060672, 0.019008, 0.091139, 0.137621, -0.060782, -0.201734, 0.176535, 0.010746, 0.027758, 0.063802, -0.154315, 0.025112, 0.075855, -0.024990, 0.008776, -0.018731, -0.047184, 0.069359, -0.048846, -0.034041, -0.109730, -0.006136, 0.078280, 0.038236, -0.102736, -0.129746, 0.075857, -0.058843, 0.102228, 0.041781, 0.026248, -0.174709, -0.124120, 0.042226, -0.009417, 0.052672, -0.018018, -0.131004, 0.031882, -0.172214, 0.153508, -0.089861, -0.032778, 0.113787, -0.005688, -0.060428, -0.148429, -0.085293, 0.112448, -0.104117, -0.164405, -0.073227, 0.074937, 0.000449, -0.036125, 0.170167, 0.104764, 0.031930, -0.006624, 0.020685, 0.093380, -0.030700, 0.101015, -0.105542, -0.169419, 0.088932, -0.102294, 0.190503, 0.106957, -0.168297, 0.060122, -0.031399, 0.034213, 0.131348, -0.038281, 0.023367, 0.034352, 0.014539, -0.081381, -0.106841, -0.172517, -0.107177, 0.162924, -0.177585, 0.109064, 0.144810, -0.026503, 0.057818, -0.058133, -0.062346, -0.166124, 0.141673, -0.056335, -0.100578, 0.035258, 0.073488, 0.008139, -0.006264, -0.208667, -0.085409, 0.111717, 0.158645, -0.152002, -0.005284, 0.180365, 0.151493, 0.090393, -0.156432, 0.242340, -0.110211, 0.056330, -0.045121, 0.065524, 0.056486, -0.014482, 0.230839, -0.009218, -0.041561, -0.052224, 0.102284, 0.305039, -0.108934, -0.065467, -0.040294, -0.128250, 0.117849, -0.282188, 0.043201, 0.009067, -0.303100, 0.102613, 0.086013, 0.054158, 0.143830, 0.103901, 0.073873, -0.185147, -0.049789, 0.141475, -0.058239, 0.144047, 0.129198, -0.188747, 0.021814, -0.058751, 0.148669, -0.075753, 0.022584, -0.207744, -0.041594, -0.131159, 0.078023, 0.111859, -0.100973, -0.165355, 0.087024, 0.008478, -0.087899, -0.092189, 0.099022, -0.074082, 0.025102, -0.034026, -0.304062, -0.035396, -0.064247, -0.112186, -0.013183, -0.294595, -0.044922, 0.058335, -0.003625, -0.175158, -0.047133, -0.021322, -0.149962, -0.030114, 0.424412, -0.135463, -0.024985, -0.102196, -0.063222, -0.174794, -0.211335, -0.076964, 0.060967, 0.076569, 0.064899, 0.008088, 0.051060, -0.325392, 0.016818, -0.231826, 0.014867, 0.016240, 0.084911, -0.011554, -0.136610, -0.023712, -0.068726, 0.108385, 0.062365, 0.105201, 0.068402, 0.054040, -0.071933, 0.033520, -0.085423, -0.058017, 0.074754, 0.056658, -0.045241, -0.014966, -0.000487, 0.129274, -0.049599, -0.164320, 0.018535, -0.016552, -0.154614, -0.170801, 0.028542, -0.101321, -0.149596, 0.097979, -0.122709, -0.122602, 0.005138, 0.077036, 0.065047, 0.093749, -0.094662, 0.112556, 0.127899, -0.133489, -0.049705, 0.063410, 0.047548, -0.033435, 0.086716, -0.156295, 0.148093, -0.077954, 0.175266, -0.070845, -0.044560, 0.065995, 0.011608, -0.037091, -0.074157, 0.066622, -0.003268, -0.001024, -0.144928, -0.018092, -0.018367, 0.149574, -0.097862, -0.035258, -0.072759, 0.010639, -0.080999, -0.107110, 0.130274, 0.021510, -0.074122, -0.161055, -0.123192, 0.005679, -0.068112, 0.081158, -0.066659, 0.024230, 0.148348, -0.100369, -0.127569, 0.024152, -0.209251, 0.021489, 0.114848, 0.040344, 0.017226, 0.063212, 0.006253, -0.031149, -0.018583, -0.012590, -0.061784, -0.145220, 0.042704, 0.020744, 0.010406, -0.040889, -0.087847, 0.086833, 0.053048, 0.133782, 0.029078, 0.031422, -0.028900, 0.008796, 0.019859, -0.151054, 0.129007, -0.148594, 0.110348, 0.059287, 0.075696, -0.099465, -0.111384, 0.064854, -0.074153, 0.215607, 0.122286, -0.167885, -0.153147, -0.027923, 0.007305, -0.209399, 0.034951, -0.052892, -0.156745, 0.162437, 0.024410, 0.207450, 0.164435, 0.036884, 0.062684, -0.176119, 0.128642, 0.067072, 0.140794, 0.090262, -0.097811, 0.165998, -0.295515, 0.032821, -0.053820, 0.198901, 0.164521, -0.224330, 0.002268, -0.178649, 0.174828, 0.010001, 0.064955, -0.113615, 0.156053, 0.022332, -0.159000, 0.121798, -0.093807, 0.055212, 0.075326, -0.044119, -0.468004, 0.039854, 0.059551, 0.080257, 0.069609, -0.209273, -0.139600, -0.015224, 0.196250, -0.155185, -0.199110, 0.100867, -0.104147, -0.120284, 0.033865, -0.030789, -0.024389, -0.145359, -0.240417, 0.021083, -0.206870, 0.123981, 0.097221, 0.059098, 0.022651, -0.145534, -0.160287, -0.193685, -0.031645, -0.112408, 0.086234, -0.112330, 0.286746, -0.167216, 0.083428, 0.036301, -0.147750, 0.016319, 0.074369, -0.004174, -0.113598, 0.115224, -0.082982, 0.094910, 0.125268, -0.099837, -0.162996, 0.043978, -0.166131, 0.031734, -0.140129, -0.084823, -0.129930, -0.007332, -0.181556, -0.168137, -0.170980, 0.007820, -0.156041, 0.115594, -0.045039, -0.037655, -0.033800, -0.032237, -0.176200, -0.167969, 0.081771, 0.025890, 0.034687, -0.084950, -0.082846, -0.069051, 0.056204, 0.101183, 0.031297, -0.070389, -0.108829, -0.131332, -0.039945, -0.013203, 0.094187, -0.161782, 0.137499, -0.189087, -0.065585, 0.010368, 0.102106, 0.084942, -0.063287, 0.086083, 0.079179, -0.034538, -0.165522, 0.054342, -0.061502, -0.137677, 0.072690, 0.126969, -0.019082, -0.062853, -0.096311, 0.116560, -0.081099, -0.176546, -0.046001, -0.125482, -0.026651, -0.162542, -0.074992, -0.115980, -0.175340, 0.004877, -0.104124, -0.138159, 0.038935, -0.132048, -0.091678, 0.128829, 0.069664, -0.088233, 0.078796, -0.156581, -0.068330, 0.005503, -0.032583, 0.120191, -0.101861, -0.127771, -0.012565, -0.189091, -0.046681, -0.032676, 0.009208, -0.030560, -0.173268, -0.174973, 0.062498, -0.140795, -0.093938, -0.112230, -0.158227, -0.031856, -0.167074, 0.101688, -0.088157, 0.085018, 0.025619, 0.128934, -0.101638, -0.082921, 0.010024, 0.028663, 0.079109, 0.002545, 0.152349, -0.038721, 0.059192, -0.125925, 0.143395, 0.135273, 0.210812, -0.114827, -0.106059, -0.030925, 0.014252, -0.152503, -0.072312, -0.098062, 0.034568, 0.043116, -0.128445, 0.097832, 0.069894, -0.038358, -0.064917, -0.005859, 0.101158, 0.004699, -0.149660, -0.059453, 0.066928, -0.011992, -0.027467, -0.147585, 0.157061, -0.152055, -0.011442, -0.112331, 0.040627, -0.029273, -0.150973, -0.023541, -0.066872, 0.063982, -0.155803, -0.071298, 0.093227, 0.137220, -0.055760, -0.140715, -0.136821, -0.139221, -0.037984, -0.097491, -0.162818, -0.022636, -0.167611, 0.104576, 0.116828, 0.112199, 0.031106, -0.176683, -0.107107, -0.152991, -0.097338, -0.159282, -0.156604, -0.011715, -0.137107, -0.080731, -0.052707, 0.068011, 0.008385, 0.100528, 0.078794, 0.108380, 0.131906, 0.070627, 0.127556, -0.139135, -0.108419, 0.019498, -0.020978, -0.050042, 0.131207, -0.127759, -0.063222, -0.045867, 0.065709, -0.018715, 0.050919, -0.118491, 0.126293, -0.152022, 0.088131, -0.134445, 0.006740, -0.161169, 0.044426, -0.084076, 0.012286, 0.020017, 0.094415, -0.067473, 0.120985, -0.015418, -0.103188, -0.172465, 0.024621, 0.083693, -0.127755, 0.032028, 0.146148, -0.138515, -0.024122, -0.077974, -0.161476, 0.142869, -0.039337, 0.022912, -0.039113, -0.062906, 0.068822, -0.072412, -0.068296, -0.022130, 0.089933, -0.012882, -0.174550, -0.138329, -0.158868, -0.145750, 0.038480, -0.176833, 0.054246, -0.027869, -0.097884, 0.034673, 0.143230, 0.069900, -0.134301, -0.075128, 0.009705, 0.086489, 0.131670, -0.008277, 0.080043, 0.066453, 0.114069, -0.048029, 0.074319, -0.023897, -0.071911, 0.179417, -0.134361, -0.089130, -0.062949, 0.061155, 0.078610, 0.067101, -0.043615, -0.025697, 0.091950, -0.103827, -0.000084, 0.182989, -0.129934, 0.009398, -0.075427, 0.162271, -0.189607, 0.092465, -0.032788, 0.059583, -0.197201, 0.112513, 0.117201, -0.094405, 0.082835, -0.078159, -0.105500, -0.188959, -0.008084, 0.113590, -0.022225, 0.092396, 0.086356, 0.013811, 0.019451, -0.130726, 0.072617, -0.128802, -0.016026, -0.091008, 0.046316, -0.072491, 0.006326, 0.044246, -0.076032, -0.006711, -0.004253, 0.099374, 0.095698, 0.123851, -0.021533, -0.185131, 0.112975, -0.069344, -0.112667, 0.003031, 0.037336, -0.046487, -0.033121, -0.117651, 0.008455, -0.152557, -0.009110, 0.101229, -0.153989, 0.037728, -0.038620, 0.108328, -0.020199, 0.041248, 0.096766, -0.032330, 0.172503, 0.059536, 0.062883, -0.053872, 0.069993, 0.014561, -0.092065, -0.182138, 0.071043, -0.229352, -0.186920, 0.030100, -0.127668, -0.036803, -0.077199, -0.141411, -0.178690, 0.045477, -0.004925, 0.070374, 0.011799, -0.062668, -0.184300, 0.042915, -0.049400, -0.134399, 0.099679, 0.047184, 0.140600, -0.027707, -0.125789, -0.048542, -0.104849, 0.071917, 0.041712, -0.011646, -0.048924, -0.012545, 0.047318, 0.009516, -0.181833, 0.063851, -0.023995, 0.064691, 0.066809, 0.173315, 0.291700, 0.140239, 0.007376, 0.058336, -0.004471, -0.062603, 0.089795, -0.032317, -0.090283, 0.227413, 0.116841, 0.041561, 0.027441, 0.144340, 0.138318, 0.075345, -0.025752, 0.063992, 0.170452, 0.082243, 0.069098, -0.181528, -0.161533, -0.088504, -0.091393, -0.110871, 0.108141, 0.077684, 0.234619, -0.113816, 0.102123, 0.012171, 0.111252, 0.142380, 0.077022, -0.123452, 0.078214, -0.002799, 0.039496, -0.050078, -0.051842, -0.032529, 0.046346, 0.131340, 0.147443, -0.054917, -0.059855, -0.070302, -0.113503, -0.119413, 0.043294, -0.080933, -0.002271, -0.155753, -0.170141, 0.058648, 0.020205, 0.005476, -0.212491, 0.096544, 0.156596, 0.042963, 0.022148, -0.051587, -0.174625, -0.003577, 0.060470, -0.085663, 0.121358, -0.114343, 0.151683, 0.171512, 0.067651, 0.051863, -0.210042, -0.008487, -0.142501, -0.108198, 0.152600, 0.042861, 0.102697, -0.036289, -0.147598, 0.182392, 0.086682, -0.287341, 0.217928, 0.065956, -0.072149, 0.200670, 0.039153, 0.031558, -0.082857, 0.085726, 0.117349, -0.075810, -0.172970, -0.078125, -0.025848, 0.021422, -0.151938, -0.148177, -0.003341, 0.000155, 0.000254, -0.112557, -0.052454, 0.032767, 0.080035, 0.033847, 0.039634, 0.136514, -0.017346, 0.106057, 0.014561, -0.101862, 0.130987, 0.032974, 0.041162, -0.168132, 0.146436, -0.051468, 0.083066, 0.033134, 0.045758, 0.018359, 0.030538, 0.099338, 0.056145, 0.094564, 0.055626, -0.099720, 0.063454, 0.159321, -0.028611, -0.119535, 0.126407, -0.046312, -0.015786, -0.167668, -0.093620, -0.068219, 0.014518, -0.135056, -0.008190, -0.143378, -0.022646, -0.089100, -0.164576, -0.036404, 0.001623, -0.010058, 0.108054, 0.107921, 0.107657, 0.045292, 0.129169, -0.005626, -0.177599, -0.010751, 0.087251, 0.089479, -0.011018, -0.015495, -0.096677, -0.057748, -0.137633, 0.108185, -0.080570, -0.027494, 0.042073, -0.069564, -0.048871, 0.060565, -0.074989, -0.094260, -0.148792, 0.002355, -0.125582, 0.128100, -0.125358, 0.004456, -0.092814, 0.046745, -0.036168, -0.063917, 0.014915, -0.108874, 0.074778, -0.119357, 0.093871, -0.053655, -0.082249, 0.091468, 0.022868, 0.129061, 0.021273, 0.085816, -0.070399, -0.061288, -0.157576, -0.078499, 0.153013, 0.111011, -0.065305, 0.154686, 0.132495, 0.059542, -0.073805, -0.061599, 0.104134, 0.132922, -0.115592, -0.031399, -0.084267, -0.053501, -0.095946, -0.019779, -0.071229, 0.063409, -0.078955, 0.149504, 0.042608, -0.028163, -0.134099, 0.109106, -0.039803, 0.045457, -0.010205, -0.214829, 0.064272, -0.063138, -0.091021, 0.119256, 0.171153, 0.143725, 0.129120, 0.060725, 0.242337, 0.144221, 0.159961, 0.102299, 0.156302, -0.073084, 0.049169, -0.006106, -0.024699, 0.075991, -0.039849, -0.152429, 0.091427, 0.152737, -0.025746, -0.049788, 0.115015, -0.137371, -0.107836, -0.175332, 0.081417, 0.079342, 0.126642, 0.089512, 0.149321, 0.054066, 0.123512, -0.119536, -0.186600, -0.070988, 0.048494, -0.090538, -0.069845, 0.186351, -0.022836, -0.035861, 0.087947, -0.057315, -0.143386, -0.137499, 0.035816, -0.035899, -0.071461, -0.020277, -0.140725, 0.085682, -0.010308, -0.093246, -0.027192, -0.004080, 0.008628, -0.065104, -0.111282, 0.076714, 0.055324, 0.043610, 0.153519, 0.015587, 0.070462, -0.019324, 0.113924, -0.084030, -0.108780, -0.109952, -0.029587, 0.042420, -0.007332, -0.001021, -0.014819, -0.103281, -0.016858, -0.098830, 0.038285, 0.077372, -0.131115, -0.131174, 0.192577, -0.035139, 0.046116, 0.008388, 0.026155, -0.078675, 0.115083, -0.173255, -0.097155, -0.122116, 0.009809, -0.094887, 0.011862, -0.008114, -0.026605, 0.094946, -0.091366, -0.043999, -0.118686, -0.021972, 0.047756, 0.084571, -0.081173, 0.105114, -0.126849, -0.079123, 0.061777, -0.028199, -0.031936, -0.042113, 0.021224, -0.011000, 0.091791, -0.102118, -0.038546, -0.068938, -0.093157, 0.098619, -0.044404, 0.030723, -0.133214, -0.044783, -0.047947, 0.100230, -0.109486, 0.070557, -0.104585, 0.096264, -0.008232, 0.071981, -0.182134, 0.074215, -0.128286, -0.024195, -0.044457, 0.038079, -0.148293, 0.009237, -0.125603, -0.022171, -0.065587, 0.103539, 0.100287, 0.021486, 0.023466, -0.142596, -0.078361, -0.124479, 0.023185, 0.106192, -0.042633, -0.027389, 0.097132, 0.086067, 0.072719, -0.098989, -0.094285, -0.163730, -0.105325, 0.211786, 0.037293, -0.074304, -0.079791, 0.083538, 0.128975, 0.031557, 0.105586, 0.081261, 0.074459, 0.083817, 0.059500, 0.110485, 0.084990, -0.004531, 0.030779, 0.035568, 0.092313, 0.141222, -0.107690, -0.046530, 0.037334, -0.004900, 0.047675, 0.041389, -0.028829, -0.146759, -0.023245, 0.150062, -0.281511, -0.048156, -0.149000, -0.025270, 0.116125, 0.020005, 0.100482, -0.187642, -0.055725, 0.041449, -0.051750, -0.055884, 0.078113, 0.062243, -0.094259, -0.131073, -0.023077, -0.061461, 0.028378, -0.120388, -0.212477, 0.122402, 0.052038, 0.059666, -0.112667, -0.076321, -0.054567, -0.058448, -0.027940, -0.011350, -0.040186, 0.059161, -0.097593, -0.156063, -0.013806, -0.117933, -0.015454, -0.184041, -0.069177, 0.024396, -0.132391, 0.182595, 0.108351, 0.001256, 0.134581, 0.065973, -0.090913, -0.024065, 0.176359, -0.004110, 0.083043, -0.068051, 0.091330, -0.029746, 0.085870, 0.011481, 0.117562, -0.176341, 0.110853, 0.020101, 0.066699, -0.044086, -0.038224, -0.043751, 0.068593, -0.092342, 0.022171, 0.094978, -0.021474, -0.068846, -0.167389, -0.099949, -0.147552, 0.109032, 0.099439, -0.105319, -0.115695, 0.020631, 0.044457, -0.104275, 0.242185, -0.089360, -0.071888, -0.107059, -0.110947, -0.041090, -0.191031, -0.032170, 0.072787, -0.048123, -0.042003, -0.156799, -0.159680, -0.071722, 0.009454, -0.078520, -0.020557, 0.032379, -0.011998, -0.138627, -0.113189, -0.043112, -0.127587, 0.186010, -0.022960, -0.159497, 0.055976, -0.010901, -0.016655, 0.095463, -0.046774, -0.114857, 0.052857, 0.129259, -0.066695, 0.111348, -0.003572, -0.095348, 0.064280, -0.180552, -0.095571, -0.021788, 0.123068, -0.007536, 0.054446, -0.196716, 0.009553, 0.021477, 0.091741, 0.005811, -0.035803, 0.148268, -0.108096, 0.156300, 0.121792, -0.106507, 0.182470, -0.051257, 0.126711, -0.159584, 0.055488, 0.078981, -0.014037, -0.059566, -0.089692, -0.132639, -0.049206, -0.064644, 0.034595, -0.076700, 0.126557, 0.104834, -0.093656, -0.100938, -0.152357, 0.020115, 0.102681, 0.106522, 0.079481, -0.021629, -0.116613, -0.170403, 0.097530, -0.123737, -0.150624, -0.100662, -0.038728, -0.082199, 0.115149, -0.100288, -0.155872, -0.027022, 0.099777, 0.081923, -0.184961, -0.011084, -0.082197, 0.136519, 0.161414, -0.176390, -0.170227, -0.082970, -0.060529, -0.066466, 0.072360, 0.036627, -0.009570, 0.029951, 0.151758, 0.056971, -0.005768, 0.181967, 0.154466, -0.115434, -0.002534, 0.014978, -0.079556, -0.175142, 0.141647, -0.138024, -0.017239, -0.004734, -0.083573, -0.084684, -0.150378, 0.012806, 0.083426, -0.179586, -0.014238, -0.112813, -0.000274, 0.102917, -0.066405, 0.009868, -0.004749, 0.115598, -0.207003, -0.044967, 0.084837, -0.120440, 0.044736, -0.038104, -0.007095, 0.018711, -0.102463, -0.098369, -0.171793, -0.070315, -0.173483, 0.067332, 0.129579, -0.013517, -0.183606, -0.141929, 0.031087, -0.135172, -0.034033, -0.027664, 0.105433, -0.063854, -0.084354, 0.148706, 0.035749, -0.201748, 0.110925, -0.108854, 0.175747, 0.109971, 0.104328, 0.067040, -0.100446, 0.084345, -0.110361, 0.110694, 0.058684, -0.154117, 0.131396, -0.128667, 0.009819, 0.077796, 0.139241, -0.012722, -0.205782, 0.068445, 0.022289, -0.120345, 0.117592, -0.033189, 0.011708, -0.025786, 0.107930, -0.071669, -0.040637, -0.171527, -0.086352, -0.081724, 0.092907, -0.095442, 0.150154, 0.023616, -0.139654, 0.030620, 0.086845, -0.079967, 0.116352, 0.032555, 0.047754, -0.093140, -0.032482, -0.139475, -0.173842, 0.146597, 0.088538, 0.030546, -0.072010, 0.092620, -0.052918, 0.070310, 0.194770, -0.001221, 0.096116, -0.044733, -0.100451, -0.157542, 0.027160, -0.163705, -0.058354, 0.085053, -0.074846, 0.099558, 0.137613, 0.131189, 0.050139, 0.091966, 0.011163, -0.165581, 0.090918, 0.074404, -0.082954, -0.170085, 0.061506, -0.004689, 0.071458, 0.131262, 0.017455, -0.081674, -0.104670, -0.072602, 0.165346, 0.106252, 0.118302, 0.107943, 0.134991, -0.157228, 0.141418, -0.132635, -0.080644, -0.019391, 0.086521, -0.052110, 0.020775, -0.166307, 0.098014, 0.144582, -0.050278, 0.013729, 0.113758, 0.149161, -0.032178, 0.028744, 0.067534, -0.156320, -0.237164, 0.117956, -0.103299, 0.085038, -0.017544, -0.139257, -0.118204, -0.032567, -0.033464, 0.085632, -0.028671, -0.075647, 0.117294, 0.164178, 0.139599, 0.085034, 0.100021, -0.163880, -0.091970, 0.021132, -0.068686, 0.178041, -0.092430, -0.120911, -0.091890, -0.052917, 0.041834, 0.215229, 0.016365, -0.160582, -0.138635, -0.002958, -0.050826, 0.087805, -0.041427, 0.226749, 0.075586, -0.016867, 0.030267, 0.094405, 0.070596, -0.039694, -0.040048, -0.171203, 0.065173, -0.013275, -0.156473, -0.078191, 0.065237, -0.078211, -0.064083, -0.169323, -0.067024, 0.172977, -0.087718, 0.002718, 0.239138, -0.037409, -0.032689, 0.055398, 0.203603, -0.040696, 0.180775, -0.042436, -0.093646, -0.137709, -0.082168, -0.018641, 0.030346, 0.139505, -0.099241, 0.019076, -0.009430, -0.024135, 0.109726, -0.167840, -0.125253, 0.026372, 0.066050, -0.213478, -0.057440, -0.046492, -0.025017, 0.073615, 0.090590, 0.009832, -0.052664, -0.136626, -0.057766, -0.011753, -0.011042, -0.060002, 0.090514, -0.115872, -0.028409, -0.112706, -0.156698, -0.156019, -0.011153, -0.041973, 0.424305, -0.068416, -0.078984, 0.059838, 0.000860, -0.002928, 0.040940, 0.041686, -0.180149, 0.029230, 0.031937, -0.031735, -0.144162, -0.263054, -0.103896, -0.111768, -0.144106, 0.046869, 0.025097, -0.057501, 0.022396, 0.129469, -0.146130, 0.146377, 0.025266, 0.023648, -0.007832, 0.059132, -0.120209, -0.069877, -0.134700, -0.035374, 0.025930, -0.118612, 0.043965, 0.100285, -0.076857, 0.056363, 0.096548, -0.083865, 0.001722, 0.133562, -0.094592, 0.047759, -0.025206, -0.045667, -0.047006, -0.015463, -0.193687, -0.170173, 0.072749, -0.028587, 0.114064, 0.003912, -0.018184, 0.005083, 0.167703, 0.054502, -0.086589, 0.132708, -0.007833, 0.118718, 0.002279, -0.074617, -0.178225, 0.100332, 0.016328, -0.098665, -0.034804, 0.145136, -0.153122, 0.075595, 0.069512, -0.178093, 0.121461, -0.160738, -0.151825, -0.069641, -0.151822, -0.012946, 0.116072, 0.057765, -0.044132, -0.136869, -0.062677, -0.021830, 0.088150, 0.064579, -0.204154, 0.023112, -0.124041, -0.074158, -0.102018, -0.026701, 0.002164, 0.090063, -0.078729, 0.016780, 0.012780, -0.006753, 0.035758, -0.073706, -0.168814, -0.075191, 0.071500, -0.031240, -0.101299, 0.099787, -0.055050, -0.063295, 0.121406, -0.183628, -0.031755, 0.124156, 0.073513, -0.013279, -0.028499, 0.108742, -0.141119, -0.039746, 0.055211, -0.133802, -0.128236, -0.103919, 0.023792, 0.030942, 0.041140, -0.051020, 0.095926, 0.022336, -0.129292, 0.049302, 0.084631, 0.050963, 0.038856, -0.079093, -0.011444, -0.171489, 0.001214, -0.005479, -0.038869, -0.093548, -0.135012, -0.040982, 0.062908, -0.051875, 0.020975, 0.123814, 0.063219, 0.041785, -0.061046, -0.022163, -0.207187, -0.043712, 0.062896, 0.030570, -0.136813, 0.115126, -0.038545, -0.107215, -0.138891, 0.094217, -0.037432, -0.061192, -0.008721, -0.089564, -0.127359, 0.026787, -0.105515, -0.028157, -0.174712, -0.051749, 0.120150, 0.101870, 0.111027, 0.056720, -0.047963, 0.009069, -0.127341, -0.015849, -0.008694, 0.069894, -0.093469, 0.037385, 0.100284, 0.171342, -0.069281, -0.211502, -0.047560, 0.123443, -0.185990, 0.163249, 0.048582, -0.225927, -0.091794, 0.067731, 0.132982, 0.144535, 0.061611, -0.132968, 0.099274, -0.237690, -0.041352, -0.086365, 0.032369, -0.039811, -0.128930, -0.050165, -0.040426, 0.039935, -0.045199, -0.122795, -0.191728, -0.017178, -0.088501, -0.106268, -0.068708, -0.085994, 0.058490, -0.032557, 0.071794, -0.146487, -0.098869, 0.007430, 0.019428, -0.087065, 0.083824, 0.112059, -0.172215, -0.154245, 0.009372, -0.055950, 0.191482, -0.096479, 0.059672, -0.155195, -0.025988, 0.046566, 0.104188, 0.036870, -0.236768, -0.028407, 0.097132, 0.083683, -0.011110, -0.156901, -0.206354, 0.000915, 0.055448, -0.129574, 0.108814, -0.124419, 0.040146, 0.067850, 0.062499, 0.100240, -0.061521, 0.117985, -0.099819, 0.025508, -0.149405, -0.125350, -0.081631, -0.001171, -0.042185, -0.164363, -0.020055, -0.202688, 0.038836, 0.026619, -0.140494, -0.084368, 0.002822, 0.005575, -0.054327, -0.076785, 0.091925, -0.034764, 0.077193, 0.114772, -0.091719, 0.036718, -0.088736, 0.037375, 0.024850, 0.110049, -0.084547, 0.029418, 0.072974, -0.164644, -0.063802, 0.019807, -0.118268, 0.002463, -0.017128, -0.178669, -0.060255, -0.147569, -0.041353, -0.151707, 0.008938, 0.020962, 0.123596, 0.121158, -0.095630, 0.122947, -0.137759, 0.071741, 0.115729, -0.113738, -0.009557, -0.128254, 0.146416, -0.176786, -0.109581, -0.026542, -0.142045, -0.027680, -0.142888, 0.061683, 0.007880, -0.053844, -0.056495, 0.067584, 0.056820, -0.096003, 0.106854, 0.018469, 0.006468, 0.001579, 0.088305, -0.172974, 0.067577, -0.036628, 0.141663, -0.156259, -0.033662, 0.036073, 0.088004, -0.007147, 0.159553, 0.037820, -0.117177, 0.101867, 0.081555, -0.027555, 0.085011, 0.106492, -0.046779, -0.118597, 0.062500, -0.108252, 0.017698, 0.032601, 0.057283, -0.073093, -0.037812, 0.114072, 0.144950, -0.163243, 0.079589, -0.166918, -0.101276, 0.041735, -0.044653, 0.141713, 0.109341, -0.067617, 0.118175, 0.088758, -0.046481, 0.058840, -0.011396, 0.037469, 0.136208, 0.213283, -0.159153, 0.063288, -0.068991, -0.019618, 0.121597, -0.154410, 0.049600, -0.034020, -0.041899, 0.070632, -0.036876, 0.060078, 0.086178, 0.029811, -0.176062, -0.072599, 0.138626, -0.026489, 0.111662, 0.057773, -0.116895, 0.079679, -0.116894, -0.048347, 0.044556, -0.051685, 0.040248, -0.177855, 0.073455, 0.112849, -0.094986, 0.115733, 0.045504, -0.122013, -0.084894, 0.078858, -0.003038, 0.004030, 0.058556, -0.046798, 0.038617, -0.076265, 0.123426, 0.163264, -0.240432, 0.048998, -0.047622, 0.003882, 0.032925, 0.103007, 0.055922, 0.198677, 0.117587, -0.100227, 0.106410, 0.008865, -0.069681, 0.022514, 0.131430, -0.107542, -0.045829, 0.107409, -0.121348, 0.111315, 0.026382, 0.033657, 0.065230, 0.013314, -0.038982, 0.169180, 0.033394, -0.061956, -0.099432, 0.006838, -0.044104, -0.048252, 0.014822, 0.099745, 0.179335, -0.038951, 0.190538, -0.038095, 0.150406, -0.119740, 0.057401, 0.008283, 0.142310, -0.052640, 0.101113, 0.087306, 0.066532, -0.155447, 0.176531, -0.103940, 0.097218, 0.123393, -0.001749, -0.108502, -0.160950, 0.068733, -0.161254, -0.087264, -0.060434, 0.118671, -0.152193, -0.132345, 0.042741, 0.072164, 0.003254, -0.119041, -0.092773, 0.125635, 0.089565, 0.085725, -0.015264, -0.186190, 0.078621, -0.147455, 0.019201, 0.062452, 0.060500, 0.123571, 0.100837, -0.011025, 0.022769, -0.138056, -0.167929, -0.123471, -0.134515, 0.026600, 0.110120, -0.014327, -0.131944, 0.079126, 0.020532, -0.004907, -0.164730, 0.110840, -0.022544, 0.034002, -0.136199, 0.029096, -0.138066, 0.029111, -0.090809, -0.211917, -0.036419, -0.024338, -0.066761, 0.025400, -0.147631, 0.088643, 0.129517, -0.088963, -0.164373, -0.079433, 0.108508, 0.095344, 0.084077, -0.043963, -0.167884, -0.059521, 0.138341, 0.072299, -0.168935, 0.046229, 0.095696, -0.154043, -0.080969, 0.030214, -0.108143, -0.075024, 0.068157, 0.084340, 0.092201, -0.133035, 0.059037, 0.017589, 0.087063, 0.037674, 0.103340, -0.067107, 0.066780, -0.159842, 0.011031, -0.063283, -0.128110, 0.115333, -0.117065, -0.023171, -0.077219, 0.011876, 0.020316, -0.110584, -0.052715, -0.055964, -0.132914, -0.092078, 0.041388, 0.050663, 0.158027, -0.051806, 0.072714, -0.114016, 0.015788, -0.022676, 0.003536, -0.075723, 0.037757, -0.092115, 0.052730, -0.119501, 0.109100, -0.020523, -0.069943, 0.029970, 0.157306, 0.139172, 0.095010, 0.112507, 0.058446, 0.087241, -0.087242, -0.162300, -0.126815, 0.010062, -0.173140, 0.012622, -0.049553, -0.002537, -0.032076, 0.020152, -0.131326, -0.054932, 0.073477, 0.163333, 0.055279, -0.005295, -0.106508, -0.030223, 0.086560, -0.105057, -0.115864, 0.192594, -0.078753, -0.155730, -0.219997, 0.048234, 0.023354, 0.072480, -0.046288, -0.109493, -0.021997, 0.083215, -0.180134, -0.160774, -0.097646, 0.104492, -0.068511, 0.025541, -0.097373, -0.077934, -0.005753, 0.068104, 0.189368, 0.091036, 0.117038, 0.031520, 0.086637, -0.132580, 0.147391, 0.040754, 0.106588, 0.075605, 0.047701, 0.141534, -0.219216, -0.076910, -0.105124, -0.156101, 0.086890, 0.043917, -0.081843, -0.016515, 0.132552, 0.014020, 0.092672, 0.079568, -0.099412, 0.123655, -0.196610, -0.098074, 0.143538, -0.095479, -0.016113, 0.061401, 0.133134, 0.066969, -0.017737, 0.079213, -0.124813, 0.176553, -0.080147, -0.023214, -0.044641, 0.004192, 0.085495, -0.238418, -0.003406, -0.014293, 0.033500, 0.098822, -0.145135, 0.087710, 0.136888, -0.023970, -0.155091, 0.051870, -0.186413, 0.110072, -0.095786, -0.001486, 0.085997, 0.053767, -0.193577, 0.009688, 0.156709, -0.046808, 0.051714, 0.075419, 0.123433, -0.044408, 0.074293, 0.069411, 0.009948, -0.179908, -0.097507, -0.053619, -0.022391, -0.016434, -0.059603, -0.078129, 0.043573, -0.046878, -0.141628, -0.055636, -0.184828, 0.012502, 0.173285, 0.029101, -0.084077, -0.032257, 0.064652, 0.095880, -0.060762, 0.072392, 0.138298, -0.076087, 0.333296, 0.021134, 0.124178, -0.177451, 0.016922, 0.071701, 0.133328, -0.044290, -0.003625, -0.053609, 0.078536, 0.118993, 0.108275, 0.047208, 0.095336, -0.101402, 0.121559, -0.067063, 0.096825, 0.016687, 0.069202, -0.061022, 0.064280, 0.005099, -0.073420, 0.134678, 0.066733, -0.009935, -0.232685, 0.108960, 0.103253, 0.113546, -0.009017, -0.096381, 0.093524, -0.043563, -0.125077, 0.064269, -0.123960, 0.049085, -0.004741, -0.125403, -0.037601, -0.035211, 0.103516, -0.010832, 0.100368, -0.095845, -0.010131, 0.003928, -0.115007, -0.117036, -0.084168, 0.032671, -0.006952, 0.153851, -0.101401, -0.059488, 0.026745, -0.068858, -0.046252, -0.045014, 0.018272, -0.031629, 0.044441, 0.119146, 0.050987, -0.147123, 0.078745, -0.008698, -0.133138, 0.051791, -0.081377, -0.159007, -0.027466, 0.017890, -0.109080, -0.015980, 0.104046, -0.063361, -0.163650, -0.010925, -0.067770, 0.089639, 0.131744, 0.033214, -0.088083, 0.064655, 0.075326, -0.046024, -0.107193, -0.052231, -0.045549, -0.014172, -0.160141, -0.039244, -0.142467, -0.023450, -0.153599, 0.087636, -0.111018, 0.160624, -0.191739, -0.168879, 0.047359, -0.035926, 0.007250, -0.100788, 0.100355, 0.118426, 0.075134, 0.036036, -0.002712, 0.075591, -0.107655, -0.006628, 0.002660, -0.056044, 0.099362, -0.091141, 0.038762, -0.120555, -0.161342, -0.009804, -0.198203, 0.078233, -0.105377, -0.047780, -0.069984, -0.148458, -0.073393, -0.116626, 0.108605, 0.052275, -0.092211, -0.118689, -0.164334, 0.046006, 0.021140, 0.009097, -0.061427, -0.162689, 0.155552, 0.127619, -0.034681, 0.039062, 0.173422, 0.109013, -0.046056, -0.151475, -0.114331, -0.097931, -0.067914, 0.090154, -0.245677, 0.050266, -0.059016, -0.003493, -0.243966, 0.005769, 0.070556, -0.051755, 0.024994, -0.152962, -0.069659, 0.079697, -0.035730, -0.005946, 0.055158, -0.123272, -0.148460, -0.089557, 0.111752, 0.102531, 0.055805, 0.033817, -0.142776, -0.188162, -0.187482, 0.032618, -0.117345, -0.011236, 0.084462, -0.057939, 0.022450, -0.175617, -0.007628, -0.060897, -0.016831, -0.094591, 0.029157, -0.083197, -0.052705, -0.082920, 0.167852, -0.155590, -0.077058, 0.072770, 0.103972, -0.142822, 0.083853, -0.120369, -0.024008, -0.127626, -0.056552, 0.010592, 0.101228, -0.178381, -0.022730, -0.140166, -0.159165, -0.151025, -0.217194, 0.085344, -0.036448, 0.121280, -0.092246, -0.025637, 0.131133, 0.106501, -0.057259, -0.056194, -0.053710, -0.045075, 0.082071, -0.034128, 0.064772, -0.123611, -0.136655, 0.070833, 0.051548, -0.002884, -0.167820, -0.174670, -0.099947, 0.055505, 0.017002, -0.161443, 0.048778, -0.065143, -0.126140, -0.164201, 0.016187, -0.077857, -0.013984, 0.031208, -0.174334, 0.022208, -0.032864, 0.113578, 0.080725, 0.074728, 0.075723, -0.012589, -0.186030, -0.154988, 0.046163, -0.171542, -0.012065, -0.071533, -0.148961, 0.087110, -0.003373, -0.147852, -0.014277, 0.053759, 0.133771, 0.075679, 0.075818, -0.168757, -0.097804, -0.024556, 0.125897, 0.019886, -0.071274, 0.085984, -0.141837, 0.020779, 0.037933, -0.069578, -0.200100, 0.038497, 0.040124, -0.158546, 0.110517, -0.224274, 0.066186, -0.067480, 0.100413, -0.079845, -0.067511, 0.040071, -0.006672, -0.195750, -0.165609, -0.130514, -0.075130, -0.067903, 0.066955, 0.010181, 0.015000, -0.191343, -0.142925, 0.137162, 0.031342, -0.017975, -0.022522, 0.010540, 0.088094, 0.024189, -0.020340, 0.080450, 0.049593, -0.062098, 0.107436, 0.033770, 0.067694, 0.098641, -0.072923, -0.109148, 0.116646, -0.111535, -0.196244, 0.136390, -0.148352, 0.070685, -0.156363, -0.144273, 0.012020, -0.186732, 0.086734, -0.120003, -0.133212, -0.029417, 0.051616, -0.086529, 0.150370, -0.143674, 0.014836, -0.016741, 0.061177, -0.001214, -0.071321, -0.119463, -0.055305, -0.055850, 0.151321, 0.106258, -0.157411, -0.028638, 0.137264, 0.062438, 0.107707, 0.017609, -0.149816, -0.109756, -0.051101, -0.046473, -0.055730, -0.011318, -0.142736, -0.151342, 0.009530, -0.078329, 0.141122, -0.118837, -0.006495, -0.019071, -0.060384, 0.025879, -0.111845, -0.096261, -0.108701, 0.024759, -0.102425, -0.051814, 0.131916, -0.156877, 0.115231, -0.050406, -0.053145, 0.060519, -0.027477, 0.049271, -0.117660, -0.159587, 0.071592, 0.082059, 0.065996, 0.041683, -0.054200, 0.025569, -0.065287, 0.029533, -0.045045, 0.040064, -0.152407, 0.175093, -0.042150, -0.024234, -0.159044, 0.071426, -0.147704, -0.112352, -0.117723, 0.076872, -0.122507, -0.062102, -0.085710, -0.128359, -0.047469, -0.063187, -0.009043, -0.082918, 0.093065, -0.108487, 0.074150, 0.001307, 0.027406, -0.069184, 0.009178, 0.055477, 0.027775, 0.049587, 0.073777, -0.159436, 0.028518, -0.096163, -0.132606, 0.120403, 0.096005, 0.058362, 0.105335, 0.073755, 0.070994, -0.135173, 0.112595, -0.015060, 0.147682, -0.132203, 0.114424, 0.014160, 0.070418, -0.037209, -0.114924, 0.082897, 0.049569, -0.105183, 0.018358, -0.159934, -0.027768, -0.144198, 0.085427, 0.143694, -0.163122, -0.051835, -0.114327, -0.076010, 0.125328, -0.125222, 0.019400, 0.071062, 0.032546, -0.088060, 0.022777, 0.024085, -0.103320, -0.131180, 0.124975, -0.160045, 0.005798, 0.124979, 0.132998, 0.048658, -0.114560, 0.093183, 0.026048, 0.058400, 0.012815, -0.074396, 0.073241, 0.065345, -0.130386, -0.034263, -0.160522, 0.004119, 0.116363, 0.065944, 0.114672, -0.042535, -0.024068, 0.055500, 0.074395, -0.067324, 0.080652, 0.017742, -0.186391, -0.044065, -0.065987, 0.040081, -0.079730, 0.004501, 0.084548, -0.136748, -0.106548, -0.056353, -0.163188, -0.151000, 0.032845, -0.043670, 0.086629, -0.155853, 0.052400, 0.179204, -0.132639, -0.160499, 0.150595, -0.088593, -0.027707, -0.213823, 0.101882, 0.020628, -0.143997, -0.067769, -0.072459, 0.048965, 0.072645, -0.004312, 0.101717, -0.221017, -0.051403, -0.160708, 0.099630, -0.020130, -0.201427, -0.060821, 0.037072, 0.048671, -0.193038, -0.157323, -0.018032, 0.055926, 0.054697, -0.125013, -0.094638, -0.035350, 0.108992, 0.067755, -0.068867, 0.104760, -0.104232, -0.132851, -0.037850, -0.191281, -0.118158, -0.111530, 0.155216, -0.092806, 0.075632, 0.201666, 0.098306, 0.047629, 0.045119, -0.040416, -0.206892, -0.073293, -0.129092, -0.100010, -0.034706, 0.070627, -0.027752, -0.149300, 0.001320, -0.122299, -0.092548, 0.024027, -0.022060, -0.072963, 0.113143, 0.135258, -0.153023, -0.015358, -0.141914, 0.042457, 0.032545, -0.027240, -0.196009, -0.197097, -0.022040, 0.005260, -0.231072, 0.021314, 0.099105, 0.117201, -0.174454, 0.098108, -0.150135, -0.121407, 0.123048, 0.107946, 0.121589, 0.117601, -0.043852, 0.136961, 0.086544, -0.162698, 0.079832, -0.057127, 0.057666, 0.166910, 0.079681, 0.023843, 0.059198, -0.112207, 0.143926, 0.100331, 0.025495, -0.068616, -0.167812, 0.031648, 0.130325, -0.124215, -0.083610, 0.012556, -0.121348, -0.002638, -0.163057, -0.117598, -0.089088, 0.109762, -0.110014, -0.067219, 0.026289, 0.165000, -0.021138, -0.010274, 0.013280, -0.199135, -0.257701, -0.118773, 0.201492, 0.052994, 0.052627, -0.109130, -0.037398, -0.081416, -0.105631, 0.082788, -0.142392, 0.141915, -0.106398, -0.043295, -0.018945, 0.016759, 0.115002, 0.010803, 0.071319, -0.146197, -0.143725, -0.136187, -0.170434, 0.052228, 0.192370, -0.070216, -0.111450, -0.170481, -0.056427, 0.066041, -0.031569, -0.043386, -0.043419, 0.071123, 0.080911, -0.174623, 0.141527, -0.035552, -0.165915, 0.079164, -0.091163, -0.016000, 0.077748, -0.070003, 0.027478, 0.075039, -0.056697, -0.086628, -0.163443, -0.134847, -0.099060, -0.097586, 0.036044, -0.089817, 0.039216, -0.180933, -0.127313, -0.152354, -0.045500, -0.016790, 0.007424, -0.030940, -0.095751, -0.008153, -0.109744, -0.017825, 0.132962, -0.161999, 0.067096, -0.024221, 0.029544, -0.041054, -0.154552, -0.010651, -0.221515, -0.172866, -0.048472, -0.102809, -0.030193, -0.005755, -0.054883, 0.051657, 0.025663, -0.042292, -0.120575, -0.001411, 0.055920, -0.079828, 0.095022, 0.105499, 0.023065, 0.018614, 0.067372, -0.019474, -0.082051, -0.139050, 0.086771, 0.048109, 0.051334, 0.035656, 0.074433, -0.150314, 0.159706, -0.054839, -0.181417, -0.091869, 0.064940, -0.123750, 0.130631, -0.157065, 0.043485, -0.034424, -0.156992, -0.090845, 0.079875, -0.107184, -0.156320, -0.094629, -0.075991, -0.018493, -0.029835, 0.068896, 0.148296, 0.050379, -0.178791, -0.086025, -0.115706, -0.003424, 0.071357, 0.087786, -0.116482, 0.055779, 0.117026, 0.006506, -0.166049, -0.172077, 0.028567, -0.177439, -0.056981, 0.003873, -0.088792, 0.039834, -0.087931, 0.117672, 0.016778, 0.099227, 0.064031, -0.063990, -0.088462, 0.020508, -0.115518, -0.064381, 0.087575, 0.067341, 0.020620, 0.017278, -0.172350, 0.113263, 0.088129, -0.068964, 0.035418, -0.083339, -0.110955, -0.032321, 0.087556, 0.112317, -0.029860, 0.185547, 0.111647, 0.195640, -0.147211, -0.075742, -0.062220, 0.007585, -0.082447, -0.215714, -0.040349, 0.000984, -0.232953, 0.116886, 0.047620, -0.077120, 0.107770, 0.099550, -0.007983, 0.025589, 0.114399, 0.117581, 0.034660, -0.019538, 0.079918, -0.042851, -0.112481, 0.104585, -0.087875, 0.136343, -0.019311, -0.032437, -0.081723, -0.164005, -0.099665, 0.123515, -0.150980, 0.126056, 0.185303, 0.033065, -0.161302, -0.156693, -0.109717, -0.013476, 0.036629, -0.165780, -0.273092, 0.104931, -0.138911, 0.017604, 0.169286, -0.027179, -0.189201, -0.160979, 0.115102, -0.003645, 0.031449, -0.069081, -0.103808, 0.029871, 0.123649, 0.033208, 0.065665, -0.109141, -0.121863, 0.079259, 0.084640, 0.026000, 0.184668, -0.034091, -0.123202, -0.011950, -0.135385, -0.252202, -0.006941, -0.046602, -0.209823, -0.163570, -0.075771, -0.135963, -0.031308, 0.055817, -0.148793, -0.124300, 0.045250, -0.041822, -0.077315, -0.139510, 0.125371, -0.027555, -0.082332, 0.009135, -0.177330, -0.108491, 0.028626, -0.071773, -0.135089, 0.048033, -0.173830, 0.051858, -0.035342, 0.025986, -0.142943, -0.072483, -0.176518, -0.016490, -0.105594, -0.042901, 0.019979, -0.106901, -0.082649, 0.019569, -0.030348, -0.072826, -0.162495, -0.030147, 0.030837, 0.009849, 0.045837, -0.054387, -0.091167, -0.077181, 0.092502, -0.070603, 0.036161, 0.035462, 0.037108, 0.056975, -0.043902, 0.135863, 0.190105, -0.174869, -0.014522, -0.163489, -0.058982, -0.046189, -0.044187, -0.138764, 0.037297, -0.101034, -0.021141, 0.100101, -0.029843, 0.068857, 0.013077, -0.055676, -0.137651, 0.093388, 0.016823, -0.116982, -0.077418, 0.032573, -0.001935, -0.130540, 0.073361, -0.062006, -0.004985, 0.070661, 0.016696, 0.095586, -0.073342, 0.117797, 0.054272, -0.089542, 0.006109, -0.084194, 0.002984, 0.016096, -0.050637, 0.043318, 0.020742, -0.029944, -0.089336, 0.137895, -0.067160, -0.068392, -0.165245, -0.038316, 0.065024, -0.001810, 0.158561, 0.033990, -0.052790, -0.017163, -0.020224, -0.118302, -0.159495, -0.141602, -0.129497, -0.063457, 0.192892, 0.033444, -0.191443, 0.056067, -0.076727, 0.170619, 0.082199, 0.055140, -0.029196, -0.133981, 0.100908, -0.170143, -0.071878, 0.056916, -0.084316, 0.122581, 0.168447, 0.139584, 0.082047, 0.029088, -0.032311, -0.071002, -0.053394, 0.154482, 0.047096, -0.051039, -0.181272, 0.069946, -0.053247, 0.099068, -0.180342, 0.015695, 0.061640, 0.090701, 0.081613, 0.068292, -0.069128, -0.153690, -0.074156, -0.170905, 0.032564, 0.092049, -0.172433, -0.124549, 0.080053, -0.007730, -0.124018, 0.038521, -0.190765, 0.110654, -0.003034, 0.094358, 0.060914, -0.165756, -0.105892, -0.109737, 0.117696, 0.029732, -0.001657, 0.009240, 0.062915, -0.107267, 0.139841, 0.108779, 0.059476, 0.071085, -0.146845, -0.052434, 0.000701, -0.138074, 0.101623, -0.222241, -0.177987, -0.109516, 0.031570, -0.089242, -0.032430, -0.150554, -0.121197, -0.103942, 0.035806, -0.086461, -0.250359, 0.126652, 0.071414, 0.175582, -0.105804, 0.165272, 0.090521, 0.118283, -0.061524, -0.136853, 0.120005, -0.024577, -0.112289, 0.109733, -0.085612, -0.217407, 0.100690, 0.188757, 0.086503, 0.035210, -0.139935, -0.134143, -0.078420, -0.144080, -0.064201, -0.135715, -0.118620, 0.089320, -0.142699, 0.093550, 0.054421, 0.100654, -0.029841, -0.144546, -0.089726, 0.133068, -0.083138, -0.087998, 0.054725, -0.048647, 0.101394, 0.039559, 0.050609, 0.033106, -0.119988, 0.107944, -0.065624, -0.028112, 0.004173, -0.061714, -0.021039, -0.132002, 0.096984, -0.015488, 0.049077, -0.134963, 0.061069, -0.082087, 0.069072, -0.156759, -0.216745, -0.140888, -0.061222, 0.069019, 0.125689, -0.045762, 0.097601, -0.013234, -0.026708, 0.065827, 0.122512, -0.048954, 0.033791, -0.037285, 0.011563, 0.147339, 0.047122, 0.133487, -0.179750, -0.147906, -0.092419, -0.190302, 0.130133, -0.101630, 0.096754, 0.133963, -0.007285, 0.091213, 0.020898, -0.018765, -0.024262, 0.034915, -0.058696, 0.023403, -0.177856, 0.095838, -0.024735, 0.124155, -0.186216, 0.095845, 0.113314, 0.123012, -0.064571, 0.069958, -0.057344, -0.025788, -0.051887, -0.006070, -0.105938, -0.109157, -0.000778, 0.075256, 0.043112, 0.108619, 0.062100, -0.147002, -0.158271, -0.035794, -0.202232, -0.053461, 0.000909, 0.131442, 0.103256, -0.165710, 0.023483, 0.004680, -0.009773, 0.037424, 0.109767, 0.028636, -0.187349, 0.022728, 0.144732, 0.064241, 0.085678, 0.132257, 0.134480, 0.015003, 0.011723, 0.018804, 0.135889, -0.078804, 0.011341, -0.183742, -0.018586, 0.001984, -0.173742, -0.020473, 0.089130, -0.178404, 0.142254, -0.123855, 0.034538, -0.031378, 0.061010, -0.169769, 0.074593, -0.042110, 0.006087, 0.045162, -0.137886, -0.120662, -0.093401, 0.111591, 0.065259, -0.106248, 0.029152, -0.040841, -0.066392, -0.204048, -0.163228, -0.160496, -0.018538, -0.083869, -0.125202, -0.143750, -0.115289, 0.045691, 0.086420, -0.038609, 0.122548, -0.058875, 0.050797, -0.024660, -0.089434, -0.044355, 0.031957, -0.122986, 0.033562, -0.076833, -0.181607, -0.102855, -0.040343, 0.013298, 0.111419, -0.180622, -0.048519, -0.019639, 0.131096, 0.101858, 0.053022, -0.017233, 0.014196, -0.087496, 0.135471, 0.058081, 0.030207, -0.005199, 0.048167, -0.112528, 0.016046, 0.009020, -0.136719, 0.106929, -0.073593, 0.058033, -0.091367, -0.055498, 0.005915, 0.061591, 0.005305, 0.083654, 0.047030, 0.013131, -0.085737, -0.090358, 0.041173, 0.045270, 0.063262, -0.087538, -0.082838, -0.049416, 0.021794, -0.112269, 0.018142, 0.013841, 0.066162, -0.151296, 0.088451, -0.018288, -0.065631, -0.181128, -0.096675, -0.042499, -0.050804, -0.047488, -0.134642, 0.110489, -0.102287, -0.116245, -0.057513, -0.024816, 0.097231, 0.042664, -0.023289, 0.062673, -0.037635, 0.084438, 0.021640, 0.083051, 0.077233, 0.091999, -0.208617, 0.127084, -0.006439, -0.023414, 0.047151, 0.164744, 0.033999, -0.143779, -0.051845, -0.076296, -0.049388, 0.001707, 0.012231, 0.039090, -0.179085, -0.165333, -0.134475, 0.082496, -0.063493, -0.233827, -0.054199, 0.069241, 0.046143, -0.089410, -0.170477, -0.138754, -0.163223, -0.015791, -0.162432, 0.094318, 0.082355, -0.024564, -0.152394, -0.034295, -0.065851, 0.116416, 0.105393, 0.035630, 0.017570, 0.160823, 0.015748, -0.134679, 0.137333, -0.049891, -0.006006, -0.133104, 0.079473, 0.016826, -0.170857, 0.022890, -0.102273, 0.107553, -0.104114, -0.170693, 0.136328, -0.026967, -0.061841, -0.112112, -0.022869, -0.091995, 0.009296, -0.028059, -0.107118, -0.117029, 0.111705, 0.031566, -0.000123, 0.003986, -0.061050, -0.047303, -0.071134, -0.114753, 0.008612, 0.024410, -0.183092, -0.008886, -0.046479, 0.023296, 0.085973, 0.078060, 0.057495, 0.038346, 0.063916, -0.101306, 0.045950, -0.137014, 0.109802, -0.143939, -0.044650, 0.053994, -0.087424, -0.072876, -0.083844, -0.123593, 0.153555, 0.104696, -0.124434, -0.042834, -0.018698, 0.068070, -0.191219, 0.024618, -0.003520, 0.137151, -0.025196, 0.004414, 0.031690, -0.126609, 0.037982, -0.075791, 0.086942, 0.081394, 0.026337, 0.040562, -0.051540, -0.050369, 0.029220, -0.038365, -0.150765, 0.013765, -0.093039, 0.017358, -0.098483, -0.063874, -0.038505, -0.084228, 0.156389, 0.031846, -0.123420, -0.105370, -0.133593, -0.102442, 0.008760, 0.037637, -0.127861, 0.045591, 0.095713, -0.075945, -0.090006, -0.135029, 0.052582, -0.166143, -0.021155, -0.134976, -0.061668, -0.077679, -0.102814, -0.014328, 0.035114, -0.059907, -0.033939, -0.108783, -0.002041, -0.154260, 0.089978, 0.139303, -0.115759, 0.113850, 0.027128, -0.128958, -0.032544, -0.030358, 0.092453, 0.002966, -0.141234, 0.045314, -0.119743, -0.005743, -0.197729, -0.076864, 0.005026, 0.084003, -0.293508, 0.095855, -0.029748, -0.032888, 0.094884, -0.059527, -0.080789, -0.075449, -0.018471, 0.146441, -0.132186, 0.081914, 0.071561, -0.178514, -0.016043, -0.054387, 0.030391, -0.202930, 0.093538, 0.060423, 0.026731, -0.025298, 0.100278, -0.175284, -0.184871, -0.148422, -0.094927, 0.059594, 0.028781, 0.100410, -0.151754, -0.032532, -0.069711, -0.007162, -0.110223, -0.013593, -0.094721, 0.065856, -0.018048, 0.106819, -0.054175, -0.186427, 0.105572, -0.259893, 0.001175, -0.115150, -0.187263, 0.040677, 0.098735, 0.060011, 0.035146, -0.074792, 0.118461, -0.065839, -0.097585, -0.168357, 0.112771, 0.078515, 0.104734, -0.104061, -0.125848, -0.107857, 0.034313, -0.125041, 0.022948, -0.132215, -0.034879, -0.209472, -0.022220, -0.094951, 0.073455, -0.145763, -0.048121, 0.121912, -0.035544, 0.075584, 0.063837, -0.088645, -0.031734, -0.170261, -0.006683, 0.070778, 0.029795, -0.030105, 0.053912, -0.074530, -0.053985, 0.097591, 0.011862, 0.026045, -0.049884, -0.076073, -0.158765, -0.004380, -0.115761, -0.176629, 0.117488, -0.125868, 0.054120, -0.098062, -0.109071, -0.151224, 0.064443, -0.031923, 0.005061, -0.073073, 0.107648, 0.099918, 0.108454, -0.182915, -0.107877, -0.108619, -0.139262, -0.027180, 0.068839, -0.136713, 0.026830, -0.071186, -0.102797, 0.079118, -0.095892, -0.039996, -0.143367, -0.054593, -0.176230, -0.066329, -0.045638, 0.134393, -0.002993, -0.139853, -0.113442, 0.125640, 0.011883, -0.003069, 0.138998, 0.029989, -0.011961, 0.163162, -0.008463, -0.194188, 0.010023, 0.095547, -0.020112, -0.116114, 0.103649, 0.118716, -0.086704, 0.037735, 0.131690, -0.079091, -0.133434, 0.021484, -0.108681, 0.018255, -0.034037, 0.065880, 0.237731, -0.140028, 0.025760, -0.065781, 0.043128, -0.016810, 0.084538, 0.076365, -0.144377, -0.114493, 0.059997, -0.160521, -0.040843, 0.049096, -0.061886, 0.060316, 0.129212, -0.101253, -0.094777, 0.003475, -0.079437, 0.099644, 0.028680, -0.134757, 0.149439, -0.154230, -0.040041, -0.207426, -0.123035, -0.027037, 0.112691, -0.023801, -0.105879, 0.131542, -0.045805, -0.090283, -0.058057, -0.166918, 0.010695, -0.168605, 0.123233, -0.161713, 0.012488, -0.112481, -0.166792, -0.167929, 0.079906, 0.015860, 0.001413, -0.010966, -0.154298, -0.016496, 0.274790, -0.063019, 0.111948, 0.051313, -0.216217, -0.082606, -0.068201, -0.101255, 0.106821, 0.069761, 0.133470, -0.014295, 0.022273, -0.117443, 0.040783, 0.021929, 0.199266, -0.035464, 0.116944, 0.009663, -0.144348, -0.022392, -0.105098, -0.089618, 0.125708, 0.117721, -0.119949, 0.024041, -0.167224, -0.123988, -0.056044, -0.136075, 0.048091, -0.002037, -0.085756, -0.136384, 0.040387, 0.060095, -0.036017, -0.003494, 0.083600, 0.023893, -0.144642, 0.011606, 0.134955, -0.121405, 0.152084, -0.171662, -0.167561, -0.052790, 0.012435, -0.115299, -0.157052, -0.169559, -0.010584, 0.051385, 0.171887, -0.048589, -0.041595, -0.198166, 0.156319, -0.038171, -0.165505, 0.021414, -0.188187, -0.161593, -0.068095, 0.072252, -0.096961, -0.031143, 0.038154, -0.187518, 0.024591, -0.064760, 0.056499, 0.040092, 0.081236, 0.134041, -0.087853, 0.084996, -0.116403, 0.008730, -0.076361, 0.113082, 0.084816, 0.048693, -0.093889, 0.040999, 0.011288, -0.075064, 0.037818, 0.047350, -0.102334, 0.108826, 0.028768, -0.096307, -0.054049, 0.006127, -0.156437, -0.011888, -0.088336, -0.017930, -0.067543, -0.182777, -0.176056, 0.079881, 0.049151, -0.031084, 0.160451, -0.084204, -0.097475, -0.013061, -0.099046, -0.024571, 0.160304, -0.190231, -0.057733, -0.165278, -0.077583, -0.084398, -0.126484, -0.012481, 0.124202, -0.177045, 0.025761, 0.097223, -0.094937, -0.083011, -0.110744, -0.016146, -0.007543, 0.128431, 0.116779, -0.188544, -0.161650, -0.100540, 0.033086, 0.101154, 0.055222, -0.158253, -0.039631, -0.060384, 0.055775, 0.048756, -0.103024, -0.081469, -0.009762, 0.072949, 0.092424, 0.113714, -0.091180, -0.015691, 0.109361, -0.078412, 0.118471, -0.113872, -0.006524, -0.167726, -0.070309, -0.138034, 0.003709, -0.050628, 0.053970, -0.093937, -0.030897, -0.125971, 0.032038, -0.030372, 0.165211, -0.129625, -0.178147, -0.144775, -0.003002, -0.151573, 0.090556, 0.112682, -0.149838, 0.042140, 0.031365, -0.195910, 0.083991, -0.108410, 0.003575, 0.063269, -0.139843, -0.004758, 0.031624, 0.060348, -0.083308, -0.073391, -0.061941, -0.061078, -0.115244, -0.016211, 0.052297, -0.084754, -0.034030, 0.075271, 0.038459, -0.081942, -0.084843, -0.047825, -0.097684, -0.174771, -0.051580, 0.088175, -0.107454, -0.090630, -0.114475, -0.141545, 0.129087, -0.038682, -0.084648, 0.135203, -0.164366, 0.191303, 0.007024, 0.229920, -0.117080, 0.138319, -0.017626, -0.039619, -0.123367, 0.091175, -0.143083, -0.029573, -0.030861, 0.085083, 0.095679, 0.111745, -0.113793, 0.081575, 0.070853, -0.071103, -0.094316, 0.127670, 0.047190, -0.038370, -0.051312, 0.183344, 0.047063, -0.126590, -0.023657, 0.095583, -0.076917, 0.008465, 0.019490, 0.006406, 0.146418, 0.058833, 0.093427, 0.172019, -0.108046, 0.168702, 0.116896, -0.081169, 0.100254, 0.099128, -0.048755, -0.099762, -0.205499, 0.067510, -0.061940, 0.121807, -0.162518, -0.065352, -0.073328, -0.147480, -0.079323, -0.044155, 0.111552, 0.142228, -0.193692, -0.094635, -0.115776, -0.146100, -0.025459, -0.158187, -0.163643, -0.064411, -0.136232, 0.080131, -0.070325, -0.071095, -0.050462, -0.133681, -0.174671, -0.005502, -0.120724, 0.009795, -0.155768, -0.186316, -0.089576, -0.145390, -0.104986, -0.087936, -0.144259, -0.121805, -0.001369, -0.137468, 0.089829, -0.098133, -0.050456, -0.187796, 0.103163, -0.148665, 0.146826, -0.028052, -0.147394, -0.094162, -0.056025, -0.090814, 0.019004, -0.116225, -0.054920, 0.030233, -0.148627, -0.200809, -0.120869, 0.101898, 0.070065, -0.117293, 0.002000, -0.191075, -0.082194, 0.036182, 0.195056, -0.159474, 0.000639, 0.010951, 0.088469, -0.021756, -0.112712, -0.121213, -0.002782, -0.106163, -0.199377, 0.013969, -0.171064, 0.057030, 0.094388, -0.093867, -0.004736, -0.115388, -0.012468, -0.122425, 0.195757, -0.109322, -0.131916, -0.126368, -0.026294, -0.023069, -0.128622, -0.122374, 0.099268, -0.017338, 0.108686, -0.075374, -0.064282, 0.071325, 0.052948, -0.164793, -0.087402, -0.048575, 0.139274, -0.132835, 0.041451, 0.019917, -0.155805, -0.112327, 0.119397, -0.166185, -0.232745, -0.100192, -0.029208, -0.042249, -0.207486, -0.158115, 0.016770, 0.048736, -0.047985, 0.056457, 0.130727, -0.138857, -0.126694, 0.180103, -0.002972, -0.098603, 0.038275, -0.086283, -0.028433, 0.014090, -0.137552, -0.204423, 0.104414, -0.137558, -0.075828, -0.038911, -0.032616, -0.005022, -0.164531, 0.170394, -0.141964, -0.013293, -0.096268, -0.091798, -0.061236, 0.138286, -0.115333, -0.037333, 0.106010, 0.058114, 0.011452, 0.089128, -0.028118, -0.117794, 0.119291, -0.122545, -0.027061, -0.018278, -0.106781, -0.134081, -0.013498, 0.098468, -0.076922, -0.135453, 0.069498, -0.058036, -0.138410, 0.089439, 0.006600, -0.116548, -0.015419, 0.031264, -0.150387, -0.049889, 0.017083, -0.018487, -0.092388, 0.031989, -0.150457, -0.151398, -0.023225, -0.137756, -0.142882, -0.072121, -0.059116, 0.064688, 0.001542, -0.014385, 0.087322, -0.109826, -0.009045, -0.104459, 0.075937, -0.145988, 0.141313, 0.098714, 0.038335, -0.006702, -0.142492, -0.010140, -0.023375, -0.039582, 0.135730, -0.014645, 0.168820, 0.041879, -0.053345, -0.170653, 0.116583, 0.101022, -0.114108, 0.100794, 0.151952, -0.014512, 0.140088, -0.126854, 0.156287, -0.131049, -0.013453, 0.016206, 0.016541, -0.098525, 0.109964, 0.118471, -0.007855, 0.087001, 0.022604, 0.140410, -0.112258, -0.075445, 0.024942, -0.076609, 0.059642, -0.157004, 0.043949, 0.159395, -0.016594, 0.016581, 0.043853, 0.093829, 0.038170, -0.006805, 0.120022, 0.050446, 0.123426, 0.014327, 0.113257, -0.031040, -0.159979, -0.136753, -0.203078, 0.076858, 0.054259, -0.047389, -0.072740, -0.023843, -0.076741, 0.057991, -0.160191, 0.119466, -0.146169, 0.159370, -0.143128, -0.010208, 0.091682, 0.022861, 0.110113, 0.091802, 0.126048, -0.132226, -0.252910, -0.076968, 0.067230, 0.023668, 0.059608, -0.070073, -0.081246, 0.028124, 0.146628, 0.071818, -0.106846, -0.046887, 0.082537, -0.058309, -0.194853, 0.026674, -0.026898, -0.182923, -0.104310, -0.061295, -0.176509, -0.001327, -0.085359, 0.103079, -0.045514, -0.142886, -0.012326, 0.005887, -0.086935, -0.022533, -0.151639, -0.156860, 0.130541, -0.030234, -0.052190, 0.131834, 0.184306, -0.139965, 0.003317, 0.078402, -0.058456, -0.084465, 0.104013, 0.080165, -0.186021, -0.041489, -0.255655, -0.081286, 0.106814, -0.118694, 0.139840, -0.159882, -0.046066, 0.015778, 0.103388, 0.085298, -0.120033, -0.136969, -0.137862, 0.055751, 0.032548, 0.089552, 0.133430, 0.066262, -0.118220, -0.091172, -0.060061, -0.052761, -0.052124, 0.072916, -0.068544, -0.115084, 0.040345, -0.041141, -0.123193, -0.165702, 0.001022, 0.042067, -0.028335, -0.056574, -0.097150, -0.054514, -0.199697, -0.003824, -0.138318, -0.052615, 0.094160, 0.172259, 0.071041, 0.150523, 0.078597, 0.027130, -0.018234, 0.037736, 0.096238, -0.095687, -0.131751, 0.078690, -0.148870, -0.014148, 0.164821, -0.128809, -0.098405, 0.034965, 0.001396, 0.011638, -0.130268, -0.047651, -0.155980, -0.190270, -0.052778, -0.018766, 0.034849, 0.130680, 0.086460, 0.108896, 0.053721, 0.014034, -0.105560, 0.128405, 0.024610, -0.137923, -0.183116, 0.146551, 0.036103, 0.036727, -0.077601, 0.072423, -0.011632, -0.092179, -0.027429, -0.096657, 0.111795, -0.007080, -0.164080, 0.059399, 0.153085, -0.019877, -0.031629, 0.000992, 0.114993, 0.003161, -0.168612, 0.127360, -0.043863, 0.039718, 0.061078, -0.161176, -0.023561, -0.007580, 0.081029, -0.059042, 0.003819, -0.166151, -0.002206, -0.044589, 0.009141, 0.070371, -0.053226, 0.006218, 0.052025, 0.112386, 0.008784, -0.124569, -0.102377, 0.052453, 0.162047, -0.125751, -0.040977, -0.049422, 0.026132, 0.054156, -0.084533, -0.024936, -0.159115, -0.050621, -0.151802, 0.045902, -0.105146, -0.148351, 0.022585, 0.029815, 0.128648, 0.094732, -0.056654, -0.142932, -0.076868, 0.143933, 0.161806, -0.148781, 0.055457, -0.066875, 0.077500, -0.171746, 0.112607, -0.026595, -0.069822, 0.017122, -0.047299, 0.128504, 0.060209, -0.004012, 0.083599, 0.037141, -0.067216, 0.054397, -0.058209, -0.052277, -0.096361, 0.047665, -0.152914, -0.103446, 0.124492, 0.051813, -0.059127, -0.066679, 0.187457, -0.183276, -0.082435, 0.018782, -0.123807, -0.058906, 0.032654, 0.014816, -0.020100, -0.132553, -0.033246, -0.120089, 0.053034, 0.046240, -0.092744, -0.122003, -0.042381, -0.144038, 0.022403, 0.146442, -0.039341, 0.020256, 0.120762, -0.079001, -0.128648, 0.107343, -0.124694, -0.008338, 0.091299, -0.179640, -0.006110, -0.070616, 0.115454, 0.058694, -0.053250, 0.020107, -0.143999, -0.061006, -0.007899, 0.096932, 0.051829, -0.093502, -0.065358, -0.075527, -0.003182, -0.128601, 0.120064, -0.069552, 0.007929, -0.080535, -0.020687, 0.047355, 0.007907, -0.134266, -0.040093, -0.097711, -0.189940, -0.084375, -0.100856, -0.124836, -0.161531, -0.122682, 0.104318, -0.125035, 0.068155, -0.007683, -0.072120, -0.159943, 0.150623, 0.078594, -0.005746, 0.010969, 0.168029, 0.154893, -0.175462, 0.149531, 0.077483, -0.150512, -0.093825, 0.050524, -0.052988, -0.137162, -0.125344, -0.008806, 0.085930, 0.052528, 0.032970, 0.040253, 0.052099, -0.132291, 0.015761, -0.060999, -0.021971, 0.110162, 0.028516, 0.103569, -0.142206, 0.006954, 0.082233, 0.020383, -0.074106, 0.024238, 0.161571, 0.092186, 0.071720, 0.020363, 0.134706, 0.110886, 0.103817, 0.002715, 0.015080, -0.114874, 0.037089, -0.081042, 0.111393, -0.010903, -0.007373, -0.104673, 0.160472, -0.047080, 0.116845, -0.091141, -0.112801, -0.131174, 0.077429, -0.064657, -0.102858, -0.031465, -0.001432, -0.010932, 0.074737, -0.055815, 0.039737, -0.066849, -0.093506, 0.099508, -0.089635, 0.086598, -0.010182, 0.028219, 0.125700, 0.043042, -0.027393, 0.050623, -0.144288, 0.011231, -0.090312, 0.094179, 0.079364, -0.058520, 0.095188, -0.061997, -0.055006, -0.109725, -0.074564, 0.045101, 0.122949, -0.081796, -0.126185, 0.109872, 0.067342, 0.145984, -0.135108, -0.069839, 0.109656, 0.094696, 0.041264, -0.056317, -0.073568, 0.038487, 0.028447, 0.055031, 0.031188, 0.093296, -0.004373, -0.011931, 0.136933, -0.130696, -0.074021, -0.172000, 0.072616, -0.092965, 0.072426, -0.069563, 0.170249, 0.060891, 0.131072, 0.051608, 0.110199, -0.160612, 0.107544, -0.007581, -0.089273, 0.086832, -0.103801, -0.173711, 0.096738, -0.016001, 0.099121, -0.126566, -0.130562, -0.197387, 0.023438, -0.133942, -0.026178, 0.040223, 0.113715, 0.051049, 0.070733, 0.091693, -0.016469, -0.009355, 0.047018, 0.130550, 0.133461, -0.308575, 0.007916, -0.155092, 0.057857, 0.019264, -0.068807, -0.086177, 0.100601, -0.145001, 0.088819, 0.011553, 0.097072, 0.047536, -0.096719, 0.011546, -0.113179, -0.083452, 0.120166, 0.077529, -0.179780, -0.005432, 0.048514, 0.102066, 0.145312, -0.125041, -0.062758, -0.162247, -0.184557, 0.059239, 0.053684, -0.021925, 0.091208, -0.214959, 0.129662, 0.066598, -0.204189, -0.169134, 0.095806, -0.008529, 0.041122, -0.060678, -0.126448, 0.034802, 0.161061, 0.046149, -0.071321, 0.132310, 0.064908, -0.147325, -0.103302, -0.044157, -0.102746, -0.168908, -0.016477, -0.093370, -0.028693, -0.120024, 0.103485, 0.095519, 0.035169, -0.009303, -0.125767, -0.192811, -0.163155, -0.159799, -0.008075, -0.054974, -0.156465, 0.103554, 0.074557, -0.105597, 0.069392, 0.106751, -0.048972, -0.044470, -0.068414, 0.163106, 0.074156, -0.113021, 0.121783, -0.002623, -0.009526, 0.031974, 0.147868, -0.065879, 0.117386, -0.122647, 0.021162, -0.038610, -0.058493, -0.029487, -0.130591, 0.060583, -0.031529, 0.010967, 0.101829, -0.162823, 0.074256, -0.005416, -0.188277, -0.086825, -0.104877, -0.046991, -0.007180, -0.116047, 0.129485, 0.028682, 0.085115, -0.091116, -0.159539, -0.018358, -0.137405, 0.039852, 0.036662, -0.121684, -0.026176, -0.037810, 0.037148, 0.009500, -0.130497, 0.071083, -0.197238, 0.069635, -0.187058, -0.100569, -0.084492, 0.164039, -0.131417, -0.032439, 0.115487, 0.082337, -0.064947, -0.108489, -0.160050, -0.108997, 0.021385, 0.062560, 0.059861, -0.050528, -0.148571, 0.092545, 0.029889, -0.122661, 0.027860, -0.015082, 0.094421, -0.182099, 0.033620, 0.023387, 0.219734, -0.053113, 0.128801, 0.044093, 0.144168, -0.098759, 0.038411, 0.126058, 0.012316, 0.137046, 0.094461, 0.025892, 0.006124, 0.014199, 0.085828, 0.026895, -0.039593, -0.097556, -0.055332, -0.006609, -0.178384, 0.021570, -0.020897, 0.267838, -0.195088, -0.148294, 0.073342, 0.016733, 0.068520, -0.139527, 0.038836, -0.060451, 0.079450, -0.166910, 0.063258, 0.068567, 0.012154, -0.077455, 0.019278, 0.044782, -0.162586, -0.122554, -0.158126, 0.118017, -0.142385, 0.055983, 0.027793, 0.104659, 0.116727, -0.017662, 0.107088, -0.181153, 0.120025, -0.094267, -0.104996, -0.100269, 0.074066, -0.122045, -0.048268, -0.153954, 0.083483, -0.056028, -0.119356, 0.069077, -0.051205, -0.114216, -0.019024, -0.061506, 0.042717, 0.028183, 0.045297, -0.074733, -0.024144, 0.048918, 0.195014, -0.038612, -0.069704, 0.181659, 0.112150, 0.046426, 0.066322, -0.067568, 0.014273, 0.015025, 0.107625, 0.076076, 0.036945, -0.093808, 0.145405, 0.150408, -0.063390, -0.167354, 0.132657, -0.002798, 0.284516, -0.234244, -0.090059, -0.174952, -0.050041, 0.166639, -0.113122, 0.004383, 0.131758, -0.172580, -0.139918, 0.102372, 0.101073, 0.160026, 0.094682, 0.114435, 0.020626, 0.001277, -0.242096, -0.047841, 0.068047, 0.087431, 0.156387, -0.141099, 0.140587, -0.096288, -0.072581, -0.155929, -0.076982, -0.063658, -0.099982, 0.003965, -0.136340, -0.104112, -0.021013, -0.060226, 0.018412, -0.058060, -0.015418, 0.068330, 0.100672, 0.127401, 0.007774, -0.165498, 0.055972, -0.032780, 0.010269, 0.050616, 0.018795, -0.095191, 0.011846, -0.090630, 0.001623, 0.003721, -0.067906, 0.120344, -0.021691, 0.045540, -0.030706, 0.183577, 0.107648, -0.259427, 0.095715, 0.043997, -0.098449, -0.073071, 0.052279, -0.059086, 0.021767, -0.154119, -0.011775, -0.060262, -0.088841, 0.051979, -0.044097, -0.058798, 0.035501, -0.044056, -0.059092, -0.144548, -0.021051, -0.091393, -0.151372, -0.151972, 0.005895, -0.054011, -0.223634, -0.174926, -0.147139, 0.093027, -0.079959, 0.061027, 0.103925, -0.014049, -0.071136, -0.006592, -0.114600, 0.079161, 0.130646, 0.032842, 0.174055, 0.043575, -0.058608, -0.130272, -0.045159, 0.137406, 0.025344, 0.128403, 0.127153, -0.076844, 0.144768, 0.051858, 0.058325, -0.006170, -0.079774, 0.128635, -0.159884, 0.012508, -0.016572, -0.164504, 0.020901, 0.052365, 0.031276, -0.097629, 0.042891, 0.065593, -0.127682, -0.101932, 0.088336, 0.064451, 0.043900, 0.087158, -0.074901, 0.040894, -0.067929, -0.089362, -0.024502, -0.011658, 0.005471, 0.108790, -0.054179, -0.176221, -0.043931, -0.109449, 0.184083, -0.006358, -0.026760, 0.012373, -0.039636, -0.037450, 0.119737, -0.051753, 0.048924, -0.007533, 0.018172, 0.033585, -0.143700, -0.187775, 0.113762, -0.043691, -0.149849, 0.008062, 0.013364, -0.026649, 0.044860, -0.171967, -0.143628, -0.084948, 0.060410, 0.039040, 0.056611, 0.014441, -0.174589, 0.006913, -0.070579, -0.116309, 0.104891, -0.057103, 0.059937, -0.010073, -0.114582, 0.067579, -0.131901, -0.028758, 0.136803, -0.103753, 0.071568, 0.079966, -0.029399, -0.005832, -0.099679, 0.060097, 0.061793, -0.153308, 0.137439, -0.060000, 0.032214, 0.107429, -0.007621, -0.056554, -0.109738, -0.079293, 0.072421, -0.028705, -0.031462, 0.005606, -0.147754, -0.066265, -0.071267, -0.092720, -0.072464, 0.149876, -0.004343, -0.055548, 0.025663, -0.047601, -0.183544, -0.148300, 0.070237, -0.022708, -0.110988, -0.107255, -0.089817, -0.056987, 0.130664, 0.094700, 0.034920, -0.167552, 0.150366, 0.020042, 0.052588, 0.106094, -0.049501, -0.094732, -0.015505, -0.156208, -0.149215, 0.004540, 0.000470, -0.049265, -0.136229, 0.038831, 0.041487, -0.174104, 0.120483, 0.090442, 0.213805, -0.033963, -0.046785, -0.119737, -0.095841, -0.107517, 0.000477, 0.055008, 0.137667, 0.052618, 0.079811, 0.042088, 0.073340, 0.028799, 0.097339, -0.165966, 0.041585, 0.116703, 0.083090, -0.102050, -0.082718, 0.154865, -0.045957, 0.103440, 0.121391, -0.125299, -0.114704, -0.064146, 0.113627, -0.007001, -0.008102, 0.137553, 0.107505, 0.067629, -0.103589, 0.099121, 0.089753, 0.162125, -0.075436, 0.087617, -0.129151, -0.002058, -0.082326, -0.065433, -0.033645, -0.073889, 0.063892, 0.171375, 0.116761, -0.117154, -0.142161, -0.076992, 0.040319, 0.015861, -0.158388, -0.100746, -0.209492, 0.015211, -0.155992, -0.219826, -0.163626, 0.116200, -0.036394, -0.158083, 0.056491, 0.101409, -0.008951, 0.013450, 0.031836, 0.032174, -0.037095, 0.153978, 0.043374, -0.004442, -0.068287, -0.123569, -0.099934, 0.081092, 0.028347, -0.068192, -0.113688, -0.018115, -0.145925, -0.078041, 0.059456, -0.091331, -0.190264, 0.024766, -0.032571, -0.129233, 0.061659, 0.008519, 0.122350, -0.033535, 0.088662, 0.105354, 0.134705, 0.031873, 0.124160, -0.083363, -0.086138, -0.034270, 0.107622, 0.024047, -0.188421, -0.141127, -0.007556, -0.025831, 0.054591, -0.087328, -0.069875, 0.124057, 0.069004, 0.029136, 0.104937, -0.088615, -0.171564, 0.044621, 0.076337, 0.198386, -0.029382, -0.086262, 0.005886, 0.016737, 0.079930, -0.025779, 0.123425, 0.004202, -0.018194, 0.112532, -0.057496, -0.089131, 0.131913, -0.103534, 0.107008, 0.074080, -0.107359, -0.147855, 0.125180, -0.184734, -0.121093, -0.173348, -0.024360, 0.066377, -0.087979, 0.088091, 0.065792, -0.199687, -0.028253, -0.120273, -0.084067, -0.014806, 0.003133, 0.028653, 0.074309, 0.001308, -0.288764, -0.168208, 0.010289, -0.107219, 0.084311, -0.170805, 0.073138, 0.089545, -0.057824, -0.037933, -0.009976, -0.039868, 0.125618, -0.101039, -0.158389, -0.000488, -0.021926, 0.112857, 0.130075, -0.039231, -0.120575, -0.021118, 0.080275, -0.061640, -0.132494, -0.166551, -0.175924, -0.204393, -0.040462, 0.059003, 0.073397, 0.047444, -0.160077, -0.092037, 0.140758, -0.096902, 0.083525, 0.023400, -0.021906, -0.051959, 0.139926, -0.028920, -0.056189, 0.028709, 0.026038, 0.149907, -0.036681, -0.197159, 0.144147, 0.037820, -0.120177, -0.036118, 0.083683, 0.100408, 0.134429, -0.106414, 0.096636, 0.143943, 0.094447, -0.068292, -0.051711, -0.076042, 0.130975, -0.108475, 0.054159, -0.145640, -0.107341, -0.100058, 0.045865, -0.165329, -0.194098, -0.061989, 0.091539, 0.173586, -0.059731, -0.097223, -0.131834, -0.060180, -0.007829, -0.058507, -0.157245, -0.174616, 0.000252, 0.153219, -0.021684, 0.001505, 0.002070, -0.117227, -0.137329, -0.050548, -0.117178, 0.083003, -0.049118, -0.144568, 0.106181, -0.144042, -0.034416, 0.081575, 0.157904, -0.017151, 0.092977, 0.061211, -0.098297, 0.069097, -0.163743, -0.126307, 0.082519, -0.117674, -0.156125, 0.026036, 0.071406, -0.002771, 0.031170, 0.003230, 0.153534, -0.154574, -0.141834, 0.026033, 0.117876, -0.061374, -0.014033, -0.113186, 0.005257, -0.105934, 0.022273, -0.087823, 0.089040, 0.088224, -0.100217, 0.000257, 0.133563, -0.145057, -0.011606, -0.205804, 0.047574, 0.017745, 0.014247, 0.111687, -0.056923, 0.058183, -0.055067, 0.029215, -0.130669, -0.012478, -0.136605, -0.042040, 0.067604, 0.074612, -0.055524, 0.030349, -0.091074, 0.096268, -0.122942, 0.006584, 0.090283, -0.122736, 0.032080, 0.078938, -0.127077, -0.031524, 0.016765, -0.034794, 0.012537, 0.049766, -0.021060, 0.131453, 0.079925, 0.107680, 0.058569, 0.018632, -0.010513, 0.028403, -0.092540, -0.129231, 0.016512, -0.144753, -0.075448, -0.159520, 0.058759, -0.118280, -0.009023, -0.020466, 0.104848, -0.133547, 0.149546, 0.113326, -0.171147, -0.096299, 0.192793, -0.022584, 0.069545, -0.046809, -0.131927, -0.028644, 0.123451, 0.012324, 0.080254, 0.000799, 0.129701, 0.002568, 0.007880, 0.012372, 0.038989, -0.022827, 0.007841, -0.114577, -0.096850, -0.076059, -0.101205, 0.001564, -0.176301, 0.098073, 0.047795, -0.012438, 0.156833, 0.071280, 0.007633, -0.136442, -0.215516, -0.182546, -0.095061, -0.034933, 0.047474, 0.133270, 0.114417, -0.153919, 0.062492, 0.039977, 0.175243, 0.155708, -0.122154, -0.033157, -0.057791, 0.005147, 0.044493, 0.015310, 0.102229, -0.124199, -0.211690, -0.191761, -0.012777, 0.038597, 0.145756, -0.034206, 0.143024, -0.181186, -0.172314, 0.047760, 0.008890, 0.049174, 0.105747, -0.036796, -0.064016, 0.108280, -0.130354, 0.043739, -0.047863, -0.144033, -0.099133, -0.113762, 0.029965, -0.058619, 0.117717, 0.069622, -0.015986, 0.046099, -0.164086, 0.113849, -0.102076, 0.010113, 0.030522, -0.181557, 0.173294, -0.015946, 0.057462, 0.046959, 0.127442, -0.096210, -0.048269, 0.032333, -0.171028, 0.011355, 0.063958, -0.117200, 0.069429, -0.009241, -0.040854, -0.163615, -0.020500, 0.004348, 0.088317, 0.132251, 0.155670, -0.092568, 0.050714, 0.200370, -0.110069, 0.026328, -0.089552, -0.023613, 0.084705, -0.118966, -0.115365, 0.056816, -0.130582, -0.132859, -0.086439, 0.003377, -0.000936, -0.128154, -0.031957, 0.162068, 0.041094, -0.109883, 0.045637, 0.135829, -0.008154, 0.115781, 0.019078, 0.121457, -0.020080, 0.081497, -0.028607, -0.083618, -0.056518, 0.120060, -0.091160, -0.053112, -0.117421, -0.021452, 0.081188, 0.027799, -0.103510, -0.159005, 0.004854, -0.072159, 0.096877, 0.039714, -0.160624, -0.094416, -0.132570, -0.067121, -0.080945, -0.047327, 0.133285, -0.042987, 0.036436, 0.064060, -0.131885, -0.002661, -0.074494, -0.109990, 0.111857, -0.032763, 0.056813, -0.123158, -0.007974, -0.087575, -0.039502, -0.029578, 0.085541, 0.033947, 0.110648, 0.033710, -0.164559, 0.030934, 0.037469, -0.194428, 0.097565, 0.040543, -0.156785, 0.056638, -0.075264, -0.146937, -0.146411, 0.130089, 0.032665, 0.090956, -0.056297, -0.096470, 0.032024, -0.049434, -0.012262, 0.059086, -0.104548, -0.119537, 0.118584, -0.135939, 0.059341, -0.009312, -0.069096, -0.109890, 0.032627, -0.041548, -0.075679, -0.017658, -0.000130, -0.145843, 0.094139, 0.138228, -0.103870, 0.070760, -0.096364, -0.207360, -0.083031, -0.212608, -0.010893, -0.121927, -0.121270, 0.032471, -0.124080, 0.137521, 0.107657, 0.019345, 0.031473, -0.104098, 0.043147, -0.001643, 0.158831, 0.039361, -0.097543, -0.082764, -0.196489, 0.160661, -0.145399, -0.006131, -0.030528, -0.118528, -0.064400, -0.117827, 0.031582, 0.030924, -0.038280, -0.042863, -0.048844, -0.037316, -0.039449, -0.045843, 0.095251, -0.043391, -0.021195, 0.036687, -0.158654, 0.005154, -0.008507, -0.033494, -0.142867, -0.017590, -0.144855, -0.106232, -0.098652, 0.013603, 0.002089, -0.011121, 0.009847, -0.044191, -0.015047, -0.153008, -0.187018, -0.028607, -0.097877, 0.006817, -0.092047, 0.117701, -0.067591, 0.066296, 0.093606, -0.066477, 0.119382, -0.164499, 0.051145, -0.098687, 0.087086, 0.106276, 0.005391, -0.127312, 0.107395, 0.107445, 0.060045, 0.049622, 0.118011, 0.067566, -0.030236, -0.037624, -0.005011, 0.099151, -0.100042, -0.092876, 0.143966, -0.117074, -0.070994, 0.006881, 0.122500, 0.073321, -0.095276, -0.047646, -0.139282, 0.013407, -0.162439, -0.165792, 0.013863, -0.074715, -0.055888, 0.054193, -0.034485, 0.011983, 0.082222, 0.125776, -0.179696, 0.048082, 0.046400, 0.029595, -0.066287, 0.009990, -0.020059, 0.092073, -0.088190, -0.046112, -0.077923, -0.079710, 0.015010, -0.105520, -0.036721, 0.023346, -0.005615, -0.107885, -0.171843, -0.069575, -0.011187, 0.065353, -0.175015, 0.060528, -0.058391, 0.071098, -0.124834, -0.110075, 0.065868, 0.135904, 0.121300, -0.032680, -0.115334, -0.075531, 0.095504, 0.145150, -0.092958, 0.041001, 0.081554, -0.073333, -0.050359, 0.018679, -0.120852, 0.075658, -0.064340, 0.087768, 0.131214, 0.002203, 0.032831, 0.008676, 0.079939, -0.010764, -0.121099, 0.086340, -0.092465, -0.082753, 0.039692, 0.159631, -0.101717, -0.090158, -0.067216, -0.082136, -0.158975, 0.117857, -0.043729, 0.146555, 0.017104, -0.181647, -0.159068, -0.054784, -0.098869, -0.056367, 0.047925, -0.026128, -0.085051, 0.016441, 0.011338, -0.160729, -0.048292, 0.114759, 0.098016, -0.111445, -0.107686, -0.114306, 0.140380, 0.034783, 0.041921, 0.071750, 0.075083, 0.096166, 0.127333, -0.170016, -0.086767, -0.037669, 0.084660, -0.145552, -0.063129, 0.098660, -0.086335, -0.086120, 0.119092, -0.050422, -0.162018, 0.085467, 0.061313, -0.139486, 0.075972, 0.055623, -0.046769, 0.105573, 0.029207, 0.002314, -0.156976, 0.082940, -0.002723, 0.112659, 0.134598, 0.157626, 0.062714, -0.075405, 0.105611, 0.017289, 0.060534, 0.062544, -0.034151, -0.041038, -0.136359, 0.013531, 0.111780, -0.116730, -0.110166, 0.005053, 0.019495, 0.120373, -0.086299, -0.070433, 0.022702, 0.055447, 0.127382, 0.023731, -0.153930, 0.011290, 0.099949, -0.045809, 0.034269, 0.148094, 0.051462, 0.040819, -0.063114, -0.133868, -0.016794, -0.168240, -0.065739, -0.134151, -0.103875, 0.117825, 0.022529, 0.105019, 0.053519, -0.163624, -0.097455, -0.027443, 0.116777, -0.112526, 0.028906, 0.090439, 0.054748, -0.198537, 0.086666, -0.016631, 0.009990, 0.148132, 0.092375, -0.029422, -0.064518, -0.012293, -0.076848, 0.031446, -0.043890, -0.134709, -0.002998, 0.040315, -0.081686, 0.001781, 0.030632, 0.126109, 0.095486, -0.152633, -0.167516, 0.099743, -0.109971, -0.114729, -0.069189, 0.073325, 0.084856, -0.103712, 0.076023, 0.110366, -0.163079, -0.132987, -0.057794, 0.102232, -0.001286, 0.068903, -0.100036, -0.011381, 0.036546, 0.107837, -0.065048, -0.072646, 0.025397, -0.013574, -0.093103, -0.163523, -0.164454, 0.087892, 0.003527, 0.004747, 0.125078, -0.023131, -0.038139, -0.080067, 0.024638, 0.000495, 0.105271, -0.051629, -0.056338, 0.104463, -0.083043, 0.011419, 0.078003, 0.053475, -0.213970, -0.170596, -0.162097, 0.139432, 0.115481, -0.190570, 0.069364, -0.161087, -0.191554, 0.012550, -0.143070, 0.039877, -0.023819, 0.055758, 0.049657, -0.004601, 0.129628, 0.051279, 0.004100, -0.060792, -0.062973, 0.156982, -0.036190, 0.033911, 0.037145, 0.016508, -0.044521, -0.133074, 0.097764, 0.086646, -0.119077, -0.204783, 0.076646, -0.087372, -0.045966, -0.104427, 0.005395, -0.137855, 0.001867, -0.005187, -0.047428, 0.012719, 0.100956, -0.092952, 0.051654, -0.129159, -0.179077, 0.056764, -0.086505, -0.096826, -0.155946, 0.084980, -0.021709, 0.146409, 0.011541, -0.219279, -0.109219, -0.150404, 0.109399, -0.006584, -0.056231, 0.115132, 0.045271, 0.108083, -0.099955, -0.020649, 0.084934, -0.080871, -0.007484, 0.023448, -0.006822, -0.145374, 0.078304, -0.028972, 0.077073, 0.114580, -0.060836, 0.117053, -0.065299, -0.027804, 0.002225, 0.114877, -0.031134, -0.026766, -0.087832, 0.087677, 0.000426, -0.136800, -0.060445, 0.084552, 0.085264, 0.088751, -0.017727, -0.006322, -0.057022, 0.101878, 0.046467, -0.050986, -0.202601, -0.016140, -0.050049, 0.046304, 0.076235, 0.088391, -0.081341, 0.079847, 0.107901, -0.007409, 0.008732, 0.048015, -0.026790, 0.052592, 0.144552, 0.149851, 0.125819, 0.066392, 0.002528, 0.068748, -0.057258, -0.152279, -0.100230, -0.037458, -0.000143, -0.080954, 0.117013, -0.177698, -0.155874, -0.016208, 0.053384, -0.189367, -0.121545, -0.083421, -0.157364, 0.055224, 0.018325, -0.018176, 0.160282, 0.101203, 0.115527, -0.114209, -0.063664, -0.012507, -0.138923, -0.049103, -0.013715, -0.004385, -0.022539, 0.166748, 0.199988, -0.029135, 0.086730, 0.111936, 0.161912, 0.083276, -0.198738, 0.084636, -0.005847, 0.118456, -0.204807, 0.113956, -0.018476, -0.023165, -0.193081, -0.146887, -0.199830, -0.126008, -0.034828, -0.168384, -0.004222, 0.098611, 0.076366, 0.024740, 0.027343, -0.138100, 0.008142, -0.185842, -0.125564, 0.023032, -0.173026, -0.140064, -0.066588, -0.011222, -0.116949, -0.107355, -0.084116, 0.031768, 0.123270, -0.015707, -0.052394, -0.112378, -0.069336, 0.149437, 0.062047, -0.007578, -0.067158, -0.143072, 0.094207, -0.096004, -0.142045, 0.093973, -0.055490, -0.008942, 0.087149, -0.161507, 0.110451, -0.051278, 0.033228, -0.149310, -0.167512, -0.032092, -0.099903, -0.090961, 0.011057, 0.003369, -0.167515, -0.076633, 0.055583, -0.115812, 0.043969, -0.089262, 0.096123, 0.100668, 0.062261, -0.072982, -0.036361, -0.001837, -0.005448, -0.120417, -0.086289, -0.147966, -0.041214, -0.008051, 0.048055, -0.037914, 0.092083, 0.006432, 0.190888, 0.064553, 0.013737, 0.061882, -0.168191, -0.011464, 0.124812, 0.005350, 0.041572, -0.098129, 0.203192, -0.009497, 0.019058, -0.027315, -0.058175, 0.064916, -0.016672, -0.056047, -0.009127, -0.035062, -0.148322, 0.028786, -0.017334, -0.002990, 0.133826, 0.134500, -0.089267, -0.051900, 0.059359, -0.102960, -0.200638, 0.059719, -0.043231, -0.080170, -0.144298, 0.162809, -0.180874, -0.114143, -0.155979, 0.126180, 0.036497, -0.110809, -0.112438, -0.131649, -0.107927, -0.078217, 0.002078, 0.050075, -0.017638, -0.139367, -0.009500, 0.013149, -0.074177, 0.006524, 0.013807, 0.050664, -0.111391, -0.111187, -0.185650, -0.173121, -0.077281, 0.010471, -0.196516, 0.055379, -0.138261, 0.059414, -0.004041, -0.138926, 0.109776, -0.202182, 0.121200, -0.064466, -0.201895, -0.074753, 0.024281, 0.098007, 0.147999, 0.001164, -0.165934, 0.026519, 0.143203, -0.025823, 0.015139, -0.124945, -0.144300, 0.086367, 0.039072, -0.091641, -0.040471, -0.135519, 0.149787, 0.064497, 0.070919, -0.179862, -0.182588, -0.093824, -0.130826, 0.005480, -0.078918, 0.073273, -0.070277, -0.028108, -0.062229, -0.147220, -0.104087, 0.127768, -0.071546, -0.030677, -0.172789, -0.147005, 0.192500, 0.061040, -0.150735, -0.057975, 0.117738, -0.039108, -0.154828, -0.204802, 0.094775, 0.070229, -0.083348, -0.058347, 0.057781, 0.036121, -0.048779, -0.173349, 0.070664, 0.129859, -0.111909, -0.088876, -0.012658, 0.074931, 0.135298, 0.017816, -0.122356, 0.069305, -0.057648, 0.163297, 0.101411, -0.032935, 0.010637, 0.132277, -0.161829, 0.028991, 0.138997, 0.132858, 0.116926, 0.069083, -0.162325, 0.035832, 0.108674, 0.014739, -0.059498, -0.148206, -0.035780, 0.020776, 0.006387, 0.098308, -0.051234, 0.023591, -0.115016, -0.162794, 0.058595, -0.125565, -0.117327, 0.162793, 0.055170, -0.057179, 0.061902, -0.025675, -0.132819, 0.045324, -0.112998, 0.051762, -0.050035, -0.074082, -0.191678, 0.107110, -0.050538, -0.073125, 0.039530, -0.006504, 0.067628, -0.122597, -0.020422, 0.041221, 0.074914, -0.160880, -0.102249, 0.022823, 0.000034, 0.082683, -0.120987, -0.010152, -0.096333, 0.109757, -0.165456, -0.118586, -0.085079, 0.073961, 0.144402, -0.088539, 0.051578, 0.063612, 0.055844, -0.130420, -0.045673, -0.044675, -0.032679, -0.081153, 0.082833, -0.020056, 0.028546, -0.013968, -0.031802, 0.072626, -0.115077, 0.026736, -0.063316, 0.081877, 0.017110, -0.082347, -0.010308, 0.051624, -0.019287, 0.003891, -0.137641, 0.097654, -0.050572, -0.138426, 0.051445, -0.026403, 0.048736, 0.153323, -0.084957, 0.175418, 0.077052, 0.061063, 0.158775, 0.098521, -0.017820, 0.107929, -0.123718, -0.089727, 0.010549, 0.095145, -0.203689, -0.069847, -0.024667, -0.063584, -0.003286, 0.007878, 0.068594, 0.054017, 0.029498, -0.104459, -0.070792, -0.013766, 0.086404, 0.006358, -0.018675, -0.016233, 0.033865, -0.117666, -0.067296, -0.083178, -0.063827, 0.015117, 0.001778, -0.059960, 0.117721, -0.106724, -0.054998, -0.086406, -0.024740, 0.045438, -0.018521, 0.162995, 0.128038, 0.066782, 0.076442, -0.091039, 0.076305, 0.058008, 0.049793, 0.040889, -0.040788, 0.038556, 0.092378, 0.013827, -0.097246, 0.114804, -0.115516, 0.103863, -0.025374, 0.180260, -0.097715, 0.078411, 0.112233, 0.124626, -0.071907, -0.048044, 0.183650, -0.031423, -0.117167, -0.042198, -0.155827, 0.010591, 0.149342, 0.068876, 0.103098, 0.073957, 0.053858, 0.089340, 0.187014, -0.114448, -0.111672, 0.107564, 0.029314, 0.159524, -0.309042, 0.089863, -0.061250, -0.181459, -0.007485, -0.002238, -0.161288, -0.045179, 0.145468, -0.011441, -0.049699, -0.005248, 0.077211, -0.122081, -0.150748, 0.081055, -0.073858, 0.110568, 0.069276, 0.119060, -0.005787, -0.253222, -0.136904, -0.000598, -0.038785, 0.054150, -0.001029, 0.075404, -0.187220, 0.082892, -0.166405, -0.157491, 0.098958, -0.125417, 0.042611, -0.169611, 0.100733, 0.083042, -0.094609, -0.105702, -0.176317, -0.217040, 0.052166, 0.127734, -0.183537, 0.134607, -0.146156, -0.063630, -0.154192, -0.166364, 0.023657, -0.152599, -0.046709, 0.029219, -0.006674, 0.140025, 0.005811, -0.008371, 0.118827, -0.086851, -0.146955, -0.128563, 0.035213, -0.140917, 0.040989, 0.168982, 0.112794, 0.025765, -0.089129, -0.197624, 0.001905, -0.003169, 0.013550, 0.088486, -0.047049, 0.128285, -0.163615, 0.138467, 0.129513, -0.161367, -0.066915, -0.023507, 0.011221, -0.124953, -0.124543, 0.067876, -0.089873, -0.069698, -0.041686, -0.293209, -0.097238, -0.156221, -0.165729, -0.069816, -0.058986, -0.135762, -0.216004, -0.157348, -0.178267, -0.244345, 0.047217, -0.063381, -0.051100, -0.120273, 0.086093, 0.081650, -0.036870, 0.036915, -0.071513, -0.153497, -0.047980, -0.110342, -0.011520, -0.003273, -0.107928, -0.115398, 0.074814, -0.030691, -0.154004, 0.073516, 0.126437, -0.009797, 0.050620, -0.154438, 0.083602, -0.069879, 0.105612, 0.041991, -0.109748, -0.095562, 0.057920, -0.146634, -0.064815, 0.037266, 0.125117, -0.155110, 0.066140, 0.075581, -0.084958, 0.087634, 0.050304, 0.115051, -0.002137, -0.115472, 0.056760, -0.049214, -0.132290, 0.023562, 0.001541, 0.053340, 0.039964, 0.117628, 0.041540, -0.072510, -0.129845, -0.016065, 0.102041, 0.096818, 0.080418, -0.007249, -0.094207, -0.060651, 0.057491, 0.063191, 0.057885, 0.081330, -0.127050, 0.181924, 0.075736, -0.032105, -0.089368, -0.030302, 0.139647, 0.021589, -0.111836, 0.116370, 0.019347, 0.052722, 0.091153, -0.149639, -0.073147, 0.075773, -0.058411, -0.061893, 0.071963, 0.116796, 0.083588, -0.045234, 0.099501, -0.179798, -0.051105, -0.005854, -0.006640, -0.034183, 0.101389, -0.068432, 0.000853, 0.038691, 0.124742, -0.203762, -0.103982, 0.098289, 0.116210, 0.050498, 0.114944, -0.099240, -0.141325, -0.175715, -0.157100, 0.005456, -0.157267, -0.017729, -0.082639, -0.190745, -0.116757, -0.011662, -0.139513, 0.152577, -0.073164, 0.083032, -0.008190, -0.158160, -0.150450, 0.067744, 0.157342, 0.082312, -0.002725, 0.051514, 0.173986, -0.022941, -0.008722, -0.116567, -0.252509, -0.070551, 0.116710, 0.158273, -0.007604, -0.091892, -0.148826, -0.145239, -0.122420, 0.000220, 0.038671, 0.089371, 0.164962, 0.085130, -0.125717, 0.025282, 0.077731, -0.089359, -0.134518, -0.173074, -0.008183, -0.084489, -0.194288, -0.132372, 0.067932, 0.073640, 0.011494, -0.171319, -0.058684, -0.166055, -0.082143, 0.045168, 0.027437, 0.057956, 0.042594, -0.089275, -0.104325, -0.162956, 0.073354, -0.146294, 0.148636, -0.115021, -0.136603, -0.029169, -0.007658, -0.094445, -0.184367, -0.158695, 0.099855, 0.122993, 0.112441, 0.133329, -0.155347, 0.078691, 0.029400, -0.084824, 0.030968, 0.109431, 0.143387, -0.049165, -0.064391, 0.138057, -0.168334, 0.095358, 0.107214, -0.149298, -0.089908, -0.005602, 0.133587, 0.024536, -0.175239, 0.015509, 0.090749, -0.004208, -0.016044, 0.016287, -0.071803, 0.056568, -0.096232, 0.125220, -0.116707, 0.055984, -0.017608, -0.074396, 0.100650, -0.150786, -0.110867, 0.100205, -0.128563, 0.015008, -0.069370, -0.109275, -0.163459, 0.120386, -0.070327, 0.001266, -0.106666, -0.127312, -0.094249, -0.034151, -0.022087, -0.080491, -0.131401, 0.014484, 0.037840, 0.119659, -0.095504, -0.113664, -0.015332, 0.114155, 0.121151, 0.041162, 0.117926, 0.007367, 0.124371, 0.057588, 0.112640, -0.095611, -0.051616, -0.032566, 0.063308, 0.015489, -0.011990, 0.057622, 0.031142, 0.139047, -0.130443, -0.034689, -0.182201, 0.046413, -0.069188, 0.108188, 0.064265, 0.050430, -0.119834, -0.178288, -0.020025, -0.061549, -0.016887, 0.104968, 0.023351, 0.090880, 0.067782, 0.084286, 0.020472, -0.122864, -0.135376, 0.079186, -0.161395, 0.004191, -0.105358, 0.130058, -0.130504, 0.087273, 0.119749, -0.097695, 0.093167, -0.183924, -0.116108, -0.156666, -0.126098, 0.073502, -0.131561, -0.116975, 0.123310, 0.013849, -0.173153, 0.025850, 0.124985, 0.106429, -0.066391, -0.020702, -0.035017, 0.063082, -0.075905, 0.051634, -0.083919, -0.068069, 0.092085, -0.132361, 0.088753, -0.138559, -0.163136, 0.068471, 0.101045, -0.054685, 0.064146, -0.107746, 0.017610, 0.066097, 0.059785, 0.084018, -0.072744, -0.036020, 0.135514, 0.105078, 0.073014, 0.098975, 0.072005, -0.029644, -0.067727, -0.171338, 0.043310, -0.050547, 0.005671, -0.030845, 0.130505, -0.088672, -0.158812, -0.155960, -0.033943, -0.181731, 0.031856, 0.086575, -0.137698, -0.143062, 0.008822, 0.025570, -0.165649, -0.138892, 0.110629, -0.045350, 0.035805, -0.012077, -0.193223, -0.053375, 0.125058, -0.164669, -0.038706, -0.114269, 0.089682, -0.063227, -0.053511, 0.109142, 0.045245, -0.025409, 0.040732, -0.030275, 0.011696, 0.187488, -0.200903, 0.002819, 0.078749, -0.112901, -0.137599, -0.015713, -0.154608, -0.088110, -0.153548, 0.080112, 0.112827, 0.106372, -0.136710, -0.127761, -0.020938, -0.101225, 0.086412, -0.003642, 0.056532, -0.077531, 0.127769, -0.039827, -0.014244, 0.016517, 0.091633, -0.050455, -0.142990, 0.000849, -0.129261, -0.056343, 0.022690, 0.004205, -0.051445, 0.003998, -0.019119, 0.092709, -0.142965, -0.174963, -0.145550, 0.124009, 0.013992, 0.120480, 0.046948, -0.108716, 0.072457, 0.116819, -0.014639, 0.081817, -0.004289, 0.176741, -0.128060, -0.076554, 0.149175, -0.135872, -0.193738, 0.121919, 0.126296, -0.142010, -0.045727, -0.009119, 0.086555, -0.015323, -0.122597, -0.060159, 0.025309, -0.041231, -0.147555, -0.143790, 0.033963, -0.122585, -0.022223, -0.082490, -0.079192, 0.002935, 0.048058, -0.120042, 0.018848, -0.084334, -0.181400, 0.005183, -0.101666, 0.054755, -0.105780, -0.176259, -0.104161, -0.157456, -0.133685, -0.112660, -0.176279, -0.013167, 0.125112, 0.016546, -0.068324, -0.134925, -0.117604, 0.133235, 0.008047, -0.052088, -0.185416, 0.000522, 0.089924, 0.030409, -0.141407, 0.013238, -0.090756, -0.026120, 0.131090, -0.070095, -0.167914, -0.031273, -0.039731, 0.099547, 0.013376, -0.049378, -0.027125, -0.137574, 0.102959, -0.155918, 0.107710, -0.136361, 0.029710, -0.015151, -0.138948, 0.083677, -0.010022, 0.181151, -0.161350, 0.123100, -0.123375, -0.147614, -0.083357, -0.099859, -0.107099, -0.009767, -0.222251, -0.088912, 0.097741, -0.057352, -0.084157, -0.079632, -0.111450, 0.020769, -0.090126, -0.053725, -0.125765, 0.077791, -0.113246, 0.097380, -0.134817, -0.092258, -0.007112, 0.052241, 0.049901, 0.033262, 0.101966, 0.070451, -0.023126, 0.041028, -0.029571, -0.083177, 0.024333, -0.093664, 0.139573, 0.057160, -0.053680, 0.036254, -0.046390, 0.052239, -0.101712, -0.055851, 0.089716, 0.059446, -0.057117, -0.092051, 0.006274, 0.024809, 0.103308, -0.020359, 0.055280, -0.091134, -0.005747, -0.155041, 0.021948, -0.086117, 0.043860, -0.019673, -0.057967, 0.135099, 0.060193, 0.077079, -0.114614, 0.002937, -0.154220, -0.088676, 0.080541, -0.162576, -0.039452, 0.017873, 0.096111, 0.141901, 0.009989, -0.161854, -0.145132, 0.009312, 0.153592, -0.027728, -0.126014, 0.114989, -0.126337, 0.145859, 0.157146, 0.054985, -0.075262, -0.060680, 0.050480, -0.119997, 0.000914, -0.034446, 0.003051, 0.050531, 0.188345, 0.108423, 0.009898, -0.167525, -0.057993, -0.044979, -0.070669, 0.047951, 0.174612, -0.141397, -0.140869, -0.022994, -0.126770, -0.025766, -0.007202, 0.178676, -0.196820, -0.056632, 0.107392, -0.135164, -0.007525, -0.128961, 0.049683, 0.075766, 0.028520, 0.006381, 0.009590, 0.071869, -0.048121, -0.004678, 0.013562, 0.154156, 0.034053, -0.090405, -0.032826, -0.065075, -0.163865, -0.045471, -0.106276, -0.184478, -0.107742, 0.110206, -0.184441, -0.023039, -0.194554, 0.060278, -0.205503, -0.043464, -0.106979, 0.128289, -0.047888, 0.028592, 0.104645, -0.135297, 0.094783, -0.024138, -0.120028, 0.049799, -0.114583, 0.009580, -0.074894, -0.003696, 0.094449, -0.178676, 0.003917, 0.058873, 0.098679, -0.070150, 0.138489, -0.123253, 0.258822, -0.013361, 0.137751, -0.115618, -0.081052, -0.235521, 0.045987, -0.056081, -0.029747, 0.092947, 0.154974, -0.123637, 0.005233, -0.017636, 0.033094, 0.095145, 0.107939, -0.104537, -0.104379, 0.099799, 0.063606, -0.088529, -0.090089, 0.020174, -0.106457, -0.107541, -0.086844, 0.037242, -0.062138, -0.022808, 0.117591, -0.219283, -0.136821, 0.040098, -0.175390, 0.046806, 0.059731, 0.089181, -0.104843, -0.040297, 0.029759, -0.150906, -0.104808, -0.047832, -0.074373, 0.015040, 0.125811, -0.064553, 0.028005, -0.133271, -0.033906, 0.040394, -0.097508, 0.075584, -0.182804, -0.040169, -0.081352, 0.011365, -0.012633, 0.094136, 0.143820, -0.137902, 0.062678, 0.152082, 0.022360, -0.110728, 0.102220, -0.037422, -0.147299, 0.114363, -0.135801, -0.144669, 0.041259, 0.006314, 0.106596, -0.019060, -0.148257, -0.067918, -0.058489, 0.101076, -0.040205, 0.013594, -0.077083, -0.051667, -0.084868, 0.089295, -0.128650, 0.079125, -0.012797, -0.017215, 0.038175, 0.065911, 0.076610, 0.207726, 0.136169, -0.164698, -0.013618, -0.014746, 0.043760, -0.018722, 0.064039, 0.119119, 0.160976, -0.112403, 0.057552, -0.031118, -0.027293, 0.042969, 0.054580, 0.199148, -0.193477, 0.011338, -0.146576, 0.101402, -0.033877, -0.136740, 0.110007, 0.072862, -0.037180, -0.069850, 0.033656, 0.145257, -0.220544, -0.068588, 0.057587, -0.047274, -0.174668, 0.051667, -0.149916, -0.097133, -0.124746, 0.060682, 0.053583, 0.105199, -0.063886, -0.010915, 0.206753, -0.039691, -0.039376, 0.045007, 0.001232, 0.056783, 0.007310, -0.035740, 0.053681, -0.033778, -0.062155, -0.202381, -0.112052, 0.091089, -0.064997, 0.071596, -0.251912, -0.081831, 0.099597, -0.200979, 0.053007, -0.002987, -0.102991, 0.068152, 0.101902, -0.019399, -0.001741, 0.118594, -0.114939, -0.109590, -0.175524, 0.017880, -0.108748, -0.164431, 0.164065, 0.067011, -0.100560, -0.056862, -0.112721, -0.028849, -0.005006, -0.098130, -0.103025, -0.062129, 0.085026, -0.035803, -0.057871, -0.016793, 0.198559, 0.115465, -0.163870, -0.066443, 0.057712, 0.079719, -0.023549, -0.100783, -0.206415, -0.062034, -0.003372, -0.061344, -0.075619, 0.141276, -0.147566, -0.034802, 0.044363, -0.091226, -0.012543, -0.011113, 0.088418, -0.021536, -0.042203, 0.100810, -0.103360, 0.163036, 0.052353, -0.010085, 0.103201, -0.133056, -0.052044, -0.152488, -0.104146, -0.051014, 0.223164, -0.089338, -0.054966, 0.060123, -0.137406, 0.119919, 0.101266, -0.059735, -0.004159, -0.053251, -0.085662, -0.066009, -0.146132, 0.141962, 0.040048, 0.167251, -0.118952, -0.055076, 0.009776, -0.206508, 0.094681, -0.194608, 0.080200, 0.017071, -0.166750, 0.135058, 0.048845, 0.027554, -0.076727, 0.063741, 0.128841, 0.162404, 0.010849, -0.081945, 0.047582, 0.034474, -0.029452, 0.043540, -0.135040, 0.130980, 0.031985, 0.063584, -0.209434, -0.166833, -0.019698, -0.108349, 0.148682, -0.081228, -0.070649, -0.212380, -0.178171, -0.077937, -0.020553, -0.045877, 0.017916, -0.093730, 0.023674, 0.114975, -0.106492, 0.093057, 0.087052, 0.166041, 0.138951, -0.132391, 0.098303, -0.020091, 0.097384, 0.080096, -0.158649, 0.123089, 0.183161, -0.142313, 0.006914, 0.139575, 0.104737, -0.279854, 0.052303, -0.103977, -0.109827, -0.168547, 0.115180, -0.176456, 0.015396, 0.036200, 0.026791, -0.039295, 0.092004, -0.086175, -0.009941, 0.006399, 0.129393, 0.136644, -0.053538, -0.182709, -0.071555, 0.053501, -0.121104, -0.155161, -0.143380, -0.034914, 0.087179, -0.114389, 0.087231, -0.189231, 0.034838, -0.035256, 0.116363, -0.073052, -0.064690, -0.047407, 0.096927, -0.023945, -0.080610, -0.062306, 0.012574, -0.116692, 0.112365, -0.088851, 0.025547, -0.122503, 0.129785, 0.044723, -0.034733, -0.071983, -0.114215, 0.007980, 0.016394, -0.091907, -0.017475, 0.011195, -0.012750, 0.078416, 0.149564, -0.118634, -0.063297, 0.019547, 0.041211, -0.070527, 0.113963, -0.028564, -0.022094, -0.114184, 0.015343, 0.097323, 0.048744, 0.107721, -0.090204, -0.148337, 0.118416, 0.142036, 0.014155, -0.146058, -0.107814, -0.056034, 0.028410, 0.064358, 0.123228, 0.046682, -0.097614, 0.124775, -0.027350, -0.143333, 0.049886, 0.029175, 0.069523, -0.122299, -0.097041, -0.165372, 0.031501, -0.065445, -0.065284, -0.023089, -0.137091, 0.031900, -0.145678, 0.141499, -0.154409, -0.076626, 0.162006, -0.104459, 0.050682, -0.073985, 0.115600, 0.030515, -0.196787, -0.053465, -0.110157, -0.155124, 0.098497, 0.147008, -0.041763, -0.192909, -0.133373, -0.140464, 0.089624, 0.010207, -0.036626, -0.109347, 0.046429, -0.039953, -0.138980, 0.126798, -0.125327, -0.010810, 0.146925, -0.185698, 0.106771, 0.118140, 0.126632, 0.043617, -0.017746, -0.039621, -0.056178, -0.028985, -0.062982, -0.117061, -0.051245, -0.170717, 0.037286, -0.008982, -0.063458, 0.034879, 0.080684, -0.101484, -0.072016, 0.110403, 0.104405, -0.056658, -0.176089, -0.033390, -0.033394, -0.038335, 0.104739, 0.068465, -0.071502, -0.152943, 0.006133, -0.115878, 0.007308, -0.076031, 0.044274, 0.015828, -0.136239, -0.128593, -0.138414, -0.088925, 0.100377, -0.100633, -0.075649, 0.124150, -0.171558, -0.055992, 0.103558, -0.057104, 0.043347, 0.000131, -0.065768, -0.052097, -0.138341, -0.111867, 0.046574, -0.018588, -0.039304, 0.098413, 0.097504, -0.102926, 0.144138, -0.141490, -0.080569, -0.140755, 0.081048, -0.037899, -0.238316, 0.077819, -0.049767, -0.067218, -0.114190, -0.066876, 0.139668, 0.074274, 0.008624, -0.153086, -0.011286, -0.112221, -0.004296, 0.063839, -0.111261, 0.189266, 0.036391, -0.031081, -0.015432, -0.114549, -0.042949, -0.108953, 0.120697, 0.029097, 0.048378, -0.142614, 0.040013, -0.023306, 0.124065, -0.141762, -0.148821, 0.068975, 0.091117, -0.116243, -0.022894, -0.059402, -0.044468, 0.041524, -0.163204, 0.006466, -0.120428, 0.032459, 0.015070, 0.081516, -0.025387, -0.081581, -0.020609, -0.131078, 0.043554, -0.118828, -0.040829, -0.083496, 0.041027, -0.239892, -0.064556, -0.164006, 0.146637, -0.202288, 0.059897, -0.174554, 0.112239, 0.131417, -0.018676, -0.062291, 0.139508, 0.017525, -0.047526, 0.125047, -0.098164, 0.020958, -0.152678, -0.092830, 0.024209, -0.052312, 0.114439, 0.026622, 0.139196, -0.110218, 0.032543, -0.097291, 0.024826, 0.064270, -0.145176, 0.097510, 0.117451, -0.006159, 0.085801, -0.008222, -0.131783, -0.035544, -0.035780, 0.098305, 0.065652, 0.033269, -0.128108, -0.136724, -0.134370, -0.150378, -0.223389, 0.069150, -0.110801, -0.055558, 0.034068, 0.042106, -0.214868, 0.120528, -0.022021, 0.032359, -0.064643, 0.062744, -0.002152, 0.141894, 0.088133, -0.108933, -0.116711, 0.004860, -0.096889, 0.103175, -0.093504, -0.114506, -0.069096, 0.087829, -0.029311, -0.087222, -0.219546, -0.167710, 0.072637, 0.114835, -0.104626, -0.068502, -0.124333, 0.101520, -0.192800, -0.049107, -0.049984, -0.087430, 0.082758, -0.066585, 0.010253, 0.049681, -0.026447, -0.113456, 0.096991, 0.113194, 0.085094, -0.025285, 0.059828, -0.203102, 0.018041, -0.169206, -0.028991, -0.127652, -0.087320, -0.112626, 0.013486, -0.049145, -0.183486, 0.077114, -0.082514, -0.031379, -0.010720, 0.004046, -0.104808, -0.147241, 0.079935, 0.067288, -0.082075, -0.006259, -0.085432, -0.017660, -0.188033, -0.137154, -0.158070, -0.086727, 0.029808, -0.099311, 0.085971, -0.030771, -0.087935, -0.102928, 0.030554, -0.258485, 0.045542, -0.098267, 0.003465, -0.038116, 0.088080, 0.085984, -0.001797, -0.144042, -0.091555, 0.134997, -0.007356, -0.097483, -0.062408, 0.094344, -0.003826, -0.107319, -0.009143, 0.060232, -0.141857, -0.189399, -0.147777, 0.042529, -0.114615, -0.097460, -0.080096, -0.152136, -0.031779, -0.001416, -0.020995, -0.010336, 0.008077, 0.054500, -0.195463, 0.042139, -0.004610, 0.099449, -0.130932, 0.032270, 0.065819, 0.063451, -0.168931, -0.175866, -0.099474, 0.066300, -0.010445, 0.091255, -0.018841, -0.181633, 0.076003, -0.091183, 0.006276, 0.012570, -0.014136, -0.028911, -0.227408, -0.082664, -0.185389, 0.080463, 0.011015, -0.106612, -0.202135, 0.059394, -0.050187, -0.097186, 0.015323, -0.020153, 0.029470, -0.040851, -0.152669, 0.069674, 0.015165, -0.106547, 0.118070, -0.143033, -0.099301, 0.098134, -0.081389, -0.143748, -0.042489, 0.044484, -0.016834, 0.102828, 0.122082, -0.109804, 0.032529, -0.157166, 0.037429, 0.144965, 0.037119, -0.041853, 0.077425, -0.127776, -0.173067, -0.244236, 0.051031, 0.015965, 0.064687, -0.111425, 0.101120, 0.140902, 0.141114, 0.002881, -0.086093, 0.042241, -0.150598, 0.116642, 0.011858, -0.118621, -0.176008, -0.080000, 0.196120, -0.050864, -0.150080, -0.061754, -0.046225, -0.080489, -0.135291, -0.144722, 0.078672, -0.060336, -0.118038, 0.021656, -0.099714, -0.012399, -0.126158, 0.080471, 0.104295, 0.109422, 0.121258, -0.048453, 0.121811, -0.106189, -0.113065, 0.064631, -0.016673, -0.089659, -0.149011, 0.112874, -0.008763, 0.132553, 0.126546, 0.056870, -0.081364, 0.057254, -0.177476, 0.225600, -0.084315, -0.005075, -0.068932, -0.199268, -0.034638, -0.003661, 0.145720, 0.063647, 0.107062, -0.101770, -0.115278, 0.119757, -0.201773, -0.153886, 0.030564, 0.016267, -0.028303, 0.080369, 0.004838, -0.030225, -0.018164, -0.128752, 0.120575, 0.075975, -0.061968, -0.216105, 0.104308, 0.046513, -0.048460, -0.021828, -0.095776, -0.053444, 0.091209, 0.070301, -0.107251, -0.014723, -0.091078, 0.021012, 0.128243, 0.069551, 0.164853, 0.044941, -0.035380, 0.005938, -0.123792, -0.076125, 0.103106, -0.042535, -0.101312, -0.162650, -0.024884, -0.086072, -0.124325, -0.036092, -0.033953, 0.081973, 0.014565, 0.106928, -0.147398, -0.137537, -0.000227, 0.085489, 0.000357, -0.002358, -0.130546, -0.088960, 0.078594, -0.016990, -0.050008, -0.068561, 0.013807, 0.136688, -0.044486, 0.073673, 0.157212, -0.150685, -0.033123, -0.124081, -0.093754, 0.000714, 0.100304, -0.184423, -0.175681, 0.026938, 0.110027, -0.193333, -0.079283, -0.086216, -0.032146, -0.146809, -0.115179, -0.045586, 0.073622, 0.010136, 0.035195, -0.009908, -0.149247, -0.156689, 0.074690, 0.022172, -0.057801, -0.099200, 0.019621, -0.078905, 0.119349, 0.097501, -0.058037, 0.068035, 0.038059, 0.127558, -0.033506, -0.075814, 0.084022, -0.114886, -0.107938, -0.164767, 0.118265, 0.115983, -0.133156, 0.015666, 0.043265, -0.091359, 0.030073, 0.113353, -0.146770, 0.018851, 0.127444, 0.136389, -0.026284, -0.152695, 0.020780, 0.051586, 0.068251, -0.176990, -0.074871, -0.013193, -0.109926, -0.076000, 0.036929, 0.068770, -0.054357, -0.013428, 0.066619, -0.084530, -0.050529, 0.045035, -0.066233, 0.014122, 0.017797, 0.134162, -0.029367, 0.133522, -0.179491, 0.059796, -0.196179, -0.013213, -0.045542, -0.008688, 0.150692, 0.127515, -0.032570, 0.056192, -0.057454, -0.134347, -0.187995, -0.115173, 0.067327, -0.044448, 0.025071, -0.159577, -0.139016, -0.054931, 0.060682, 0.042887, -0.134104, 0.127683, 0.071640, -0.097620, -0.041133, 0.104649, 0.052496, -0.183604, -0.142137, -0.158570, -0.117071, 0.062870, -0.182715, -0.118902, 0.023776, 0.105732, 0.067152, -0.131138, -0.060544, -0.075745, 0.122732, 0.013146, 0.111522, 0.083813, -0.079083, -0.180263, 0.173437, -0.078888, -0.110326, -0.062059, -0.217398, 0.029420, 0.042192, -0.131865, -0.040168, 0.097468, 0.022041, 0.142726, -0.024543, -0.025416, -0.057573, 0.003270, 0.062648, -0.237449, 0.055696, -0.016585, -0.035708, 0.058412, 0.118583, -0.113662, -0.171701, -0.084177, -0.086037, -0.001453, -0.056208, -0.005314, 0.079942, -0.046683, -0.081159, 0.038092, 0.039165, 0.061178, 0.050048, -0.192825, 0.092904, 0.010096, -0.160580, -0.053810, 0.110040, -0.105207, 0.022737, 0.052208, -0.197196, 0.077586, 0.074730, -0.032857, -0.022817, -0.044641, 0.096452, 0.071437, -0.040647, -0.068381, -0.149945, 0.010427, 0.095166, 0.084576, 0.056924, 0.002740, -0.060144, 0.110018, 0.123764, -0.101076, -0.115177, 0.061039, -0.058669, -0.114823, -0.018381, -0.040095, 0.109209, -0.007700, 0.054180, 0.065105, 0.154808, -0.069683, 0.157611, -0.092594, -0.009851, 0.147449, -0.140320, -0.023466, 0.000146, 0.024859, -0.064287, 0.095455, -0.223994, 0.074665, 0.128317, -0.183614, 0.031620, -0.166497, -0.113748, -0.078940, -0.079629, -0.070505, -0.032896, -0.115736, -0.233784, 0.028307, 0.048919, -0.103068, -0.125254, -0.197099, 0.088422, -0.082112, -0.150265, 0.085600, 0.145839, -0.036611, -0.038423, 0.076570, -0.102502, 0.038212, -0.058771, 0.100135, -0.112996, 0.113948, 0.078646, 0.068558, 0.000872, -0.094352, -0.085134, 0.016940, 0.049182, -0.149459, -0.040663, 0.160288, -0.058054, -0.107129, -0.027434, 0.120038, -0.042512, 0.098217, -0.056400, 0.114359, -0.138199, -0.174845, -0.046696, -0.133190, 0.149010, -0.095446, 0.086586, 0.012126, -0.129338, 0.082485, -0.149216, 0.111288, -0.157902, -0.145315, -0.166313, -0.154637, 0.034663, 0.057126, 0.017538, -0.035673, -0.075994, -0.045146, -0.075083, -0.085789, 0.110572, -0.064468, -0.097792, -0.121533, 0.004699, 0.018970, 0.090067, -0.154906, 0.128776, 0.052577, 0.272932, 0.078032, -0.115124, -0.100994, 0.080838, 0.106737, -0.010781, -0.026414, -0.085937, -0.033596, -0.032546, 0.118558, 0.037313, -0.152114, -0.020536, -0.096719, -0.038114, -0.002975, -0.179399, 0.035396, -0.113015, 0.068077, -0.117978, 0.246018, -0.255393, -0.151490, 0.112365, -0.037704, -0.146541, -0.127236, 0.033792, -0.158600, -0.076285, 0.019814, 0.000345, -0.190952, 0.012936, 0.044876, 0.082551, 0.069024, -0.015924, -0.200922, -0.194196, 0.008872, 0.040545, 0.069285, -0.178859, 0.088852, 0.087090, 0.083974, 0.028265, -0.204634, 0.120204, -0.143886, 0.019109, -0.175361, 0.000450, -0.048338, -0.032716, -0.019891, -0.204724, -0.006237, -0.015328, 0.027481, -0.095115, -0.080982, -0.131405, -0.025104, 0.119570, -0.031411, 0.002688, -0.006044, -0.001053, -0.147617, 0.091504, 0.133549, 0.064974, -0.182272, -0.039824, -0.105673, 0.117447, 0.086035, 0.059157, 0.001144, -0.033547, 0.041183, -0.017162, -0.119288, 0.008348, -0.118633, -0.080191, 0.120480, 0.123630, 0.105891, 0.077004, 0.015718, 0.074197, -0.074893, -0.024445, 0.023867, -0.108407, 0.016913, -0.081505, 0.040614, 0.068392, 0.062925, -0.113308, -0.148656, 0.025292, 0.075382, -0.128540, -0.052672, 0.102644, -0.037226, 0.042145, -0.079871, -0.021239, 0.062089, -0.080536, -0.004878, -0.028074, 0.085588, -0.070455, 0.034130, 0.121478, -0.060853, 0.001182, 0.072756, 0.184900, 0.046974, 0.007254, 0.044256, -0.076773, 0.113850, -0.064104, 0.141170, 0.140324, -0.085284, 0.170243, -0.128766, -0.061961, -0.045401, 0.093604, -0.046991, -0.054597, -0.097401, 0.058838, -0.169127, 0.098597, 0.143315, 0.024941, -0.068958, -0.017065, 0.152971, -0.153009, 0.061297, -0.072873, -0.116670, -0.047135, -0.068578, -0.038568, -0.017340, -0.136063, -0.120270, -0.000018, 0.019398, -0.048910, 0.141686, -0.169556, -0.127560, -0.088365, 0.242947, -0.012367, -0.029260, 0.112682, 0.146264, 0.035581, -0.065821, -0.120217, -0.111281, 0.047625, 0.127282, -0.124077, 0.026581, -0.032569, -0.134355, 0.001502, -0.001670, 0.130715, -0.140511, -0.092148, 0.113554, 0.126217, -0.127600, -0.154533, -0.130864, 0.151548, -0.165952, -0.093601, -0.115502, 0.111661, -0.149739, -0.005096, -0.001746, -0.105613, -0.113069, -0.091251, -0.047173, -0.082413, -0.057089, 0.034215, 0.009527, 0.050689, 0.018993, 0.098325, -0.103830, -0.028448, 0.132497, -0.106403, -0.091383, 0.093465, 0.019489, 0.107034, -0.005923, -0.107828, 0.090007, 0.078876, -0.139402, -0.148835, 0.132725, 0.055199, 0.107953, 0.112277, 0.144955, 0.017449, 0.046704, -0.039321, -0.100851, 0.080373, 0.051037, -0.021213, -0.027067, -0.010200, 0.085427, 0.109527, -0.082218, -0.031878, -0.014328, -0.037179, -0.079513, -0.045509, 0.126207, 0.134184, 0.089526, -0.134983, -0.034865, -0.130552, -0.096091, -0.039944, -0.094928, -0.091325, 0.036404, 0.067385, -0.155155, -0.053282, 0.120045, 0.001179, -0.054267, -0.064153, 0.146174, 0.109511, -0.140114, -0.044743, -0.026400, -0.006362, 0.027609, 0.056892, -0.063629, 0.055468, 0.201924, 0.147733, 0.018782, -0.031674, -0.025117, 0.092058, -0.076673, 0.066793, -0.096280, -0.080339, -0.102944, -0.200353, 0.005742, -0.107385, -0.011048, 0.218070, -0.154980, -0.030402, -0.055634, -0.095756, 0.051839, 0.041783, -0.079084, 0.057158, -0.050523, -0.191625, 0.002064, -0.035025, 0.175336, 0.004292, 0.012268, 0.085485, -0.062165, 0.054895, -0.058532, -0.006035, -0.090777, 0.161748, 0.042589, 0.003468, 0.148488, -0.177345, -0.119622, 0.103376, -0.053838, -0.375238, -0.186718, -0.003888, -0.031300, 0.146053, -0.235090, 0.046761, -0.057574, 0.102913, 0.082817, -0.157544, 0.073712, -0.060517, 0.149766, 0.013649, -0.090456, -0.151764, -0.108029, -0.017575, -0.067129, -0.132946, 0.115882, 0.191901, -0.186642, 0.105434, 0.001279, 0.052418, -0.236294, 0.228127, -0.107996, 0.141964, 0.141242, 0.112522, -0.029374, -0.115662, 0.068836, 0.088019, -0.068281, -0.122744, -0.056512, -0.160396, -0.097851, 0.082139, -0.022929, -0.097554, 0.050037, -0.050706, -0.092552, -0.151943, -0.039480, 0.098221, 0.025363, 0.121856, -0.019623, -0.050998, 0.085980, -0.103682, -0.024557, -0.028154, 0.140678, -0.134240, 0.004944, 0.171530, -0.035597, -0.059066, 0.067948, -0.136417, 0.043533, 0.085510, 0.141027, 0.089203, -0.173238, 0.024916, -0.188280, -0.078622, 0.007307, 0.001136, -0.032833, 0.136877, -0.040275, -0.107047, -0.026199, -0.111873, -0.077519, 0.060953, -0.081209, -0.089078, -0.131212, -0.214386, 0.039660, -0.007996, -0.041032, -0.143363, -0.041879, -0.128621, -0.032257, 0.089986, -0.128163, -0.147783, 0.040123, -0.054309, 0.137640, -0.113711, 0.087602, -0.020807, 0.046376, -0.117036, -0.086622, 0.073484, -0.106715, -0.008496, -0.041265, 0.032689, -0.036737, -0.023509, -0.010423, -0.097932, 0.127922, 0.092023, -0.261317, -0.037279, 0.068196, -0.043872, -0.059423, 0.118197, -0.017536, -0.165101, -0.151433, -0.062144, 0.077351, -0.111120, -0.000468, -0.171055, -0.095577, -0.081310, -0.067878, -0.106086, 0.073652, -0.085683, 0.115130, -0.023699, -0.255251, 0.009833, 0.079403, -0.046998, -0.144311, 0.045148, -0.141484, 0.039933, -0.240095, 0.024020, -0.161332, 0.072830, -0.030642, 0.095275, -0.031720, 0.080813, -0.049839, 0.132595, 0.111248, -0.128170, 0.144686, 0.106060, -0.073205, -0.112116, 0.064054, 0.124255, 0.077049, -0.103757, -0.033606, 0.057244, -0.183980, -0.113916, -0.015967, 0.158378, -0.211174, 0.058756, -0.090950, -0.020055, -0.204556, 0.004493, 0.130773, 0.044375, 0.111087, -0.095677, -0.083667, -0.120321, -0.119376, 0.099119, 0.070604, 0.216802, -0.016641, -0.089297, -0.071857, 0.088992, -0.042410, -0.166470, -0.048789, 0.159211, 0.020969, 0.027951, -0.147925, -0.095985, -0.203454, -0.099532, 0.081401, 0.086816, -0.072892, -0.014783, -0.042842, -0.018475, 0.004057, 0.061175, -0.042673, -0.115115, -0.061517, -0.181566, -0.048577, 0.078439, 0.030115, 0.096284, 0.122027, 0.015091, -0.001952, -0.184665, -0.183340, 0.121161, 0.077084, 0.120614, 0.036653, -0.041136, -0.095274, -0.076469, 0.016067, -0.152574, -0.161004, -0.053700, -0.174915, 0.055764, 0.055530, -0.047575, 0.110733, 0.038371, -0.138825, -0.005829, 0.077527, -0.097354, -0.150079, -0.138127, 0.020164, -0.137939, -0.055571, -0.051145, -0.010957, -0.050050, 0.027898, 0.128095, -0.039722, -0.163414, -0.115441, -0.140386, -0.060645, -0.143021, -0.040438, -0.073705, 0.092870, 0.025488, 0.057359, 0.035007, 0.034269, -0.184439, -0.008568, -0.036672, -0.117755, -0.078219, -0.014642, -0.003773, 0.112735, 0.159742, 0.073783, -0.102134, -0.057751, 0.100157, 0.011945, 0.111263, -0.114283, 0.142957, 0.088865, 0.008297, -0.094911, -0.108415, 0.129853, -0.026366, 0.139512, -0.054371, -0.068691, 0.011263, 0.083911, -0.142222, -0.148573, -0.180843, -0.177897, 0.101703, -0.091163, 0.115123, -0.076116, 0.121062, 0.044440, -0.004242, 0.038957, -0.098191, 0.079323, 0.149679, -0.079733, 0.134394, 0.069309, -0.029917, 0.126253, 0.135795, 0.045488, -0.071909, 0.041976, 0.072728, 0.043411, 0.095179, 0.011461, -0.084031, 0.049067, -0.027332, -0.194251, 0.092667, -0.065530, 0.015394, 0.039194, 0.078328, -0.037340, -0.081218, -0.166217, 0.079373, -0.106995, -0.072569, 0.041219, -0.092890, 0.026647, 0.113741, -0.011953, -0.015872, -0.107874, -0.061711, -0.002922, 0.064336, 0.019507, 0.061140, 0.022263, 0.104685, -0.005835, 0.067752, -0.048613, -0.061207, 0.050842, -0.058667, -0.024977, -0.022151, -0.026875, 0.070869, -0.112406, 0.015243, 0.147085, 0.103210, -0.155661, 0.100810, 0.038450, 0.007887, -0.141723, 0.008952, 0.064235, -0.057354, -0.057465, -0.109139, 0.080753, -0.203051, 0.062063, 0.013755, 0.110936, -0.071486, -0.137201, -0.150960, -0.046566, 0.002241, -0.112229, 0.139983, -0.025322, 0.133997, -0.005276, -0.038675, 0.064901, 0.035652, 0.114249, -0.176375, -0.006449, 0.028156, -0.012417, 0.087935, 0.048660, -0.008814, -0.015440, -0.139947, -0.047276, -0.075980, -0.015994, -0.063570, 0.198087, -0.015379, -0.080554, -0.067341, 0.131144, 0.025714, 0.018303, -0.097610, -0.034295, -0.008001, 0.013472, 0.041649, -0.195262, -0.148865, -0.214648, -0.120172, 0.116580, -0.139312, -0.040799, -0.090823, -0.082462, -0.189949, -0.068030, 0.097381, -0.087591, 0.122938, -0.034352, -0.190574, 0.028857, -0.118793, 0.128314, -0.088266, 0.137270, -0.064948, -0.158166, -0.034857, -0.174278, 0.021859, -0.211957, -0.230305, -0.120051, -0.155680, 0.119348, -0.186901, -0.003813, 0.091599, -0.159798, -0.106841, 0.011901, 0.054900, 0.089035, 0.124179, 0.095424, -0.039303, 0.021963, 0.067248, 0.125447, 0.015586, -0.147662, 0.142783, 0.068611, 0.072309, -0.145407, -0.123292, -0.146130, 0.054221, -0.089213, 0.067318, -0.142929, 0.086959, -0.141821, -0.045978, -0.091561, -0.011516, -0.052907, 0.083816, -0.154937, 0.005610, -0.111047, 0.022628, -0.156896, -0.080070, 0.023246, 0.011472, -0.157709, -0.075989, 0.016633, 0.090595, -0.033119, 0.088691, 0.151322, -0.210669, -0.085613, -0.036806, -0.066193, -0.082845, 0.112928, 0.048747, -0.103974, -0.088600, -0.044678, -0.034222, 0.060219, 0.136934, -0.152825, -0.181681, 0.038132, -0.055632, -0.061142, 0.038719, -0.108628, -0.033752, -0.065010, -0.118702, -0.008705, -0.103781, -0.021544, 0.052863, -0.094435, 0.058808, -0.046397, -0.027185, 0.024454, 0.016023, -0.129484, 0.080126, 0.153517, -0.186218, 0.099362, -0.049563, -0.113920, 0.076801, -0.220342, 0.125953, 0.031652, 0.041190, 0.014747, -0.150906, 0.090607, -0.036862, 0.006491, -0.134972, -0.173681, -0.110063, -0.126986, -0.118076, -0.146544, 0.060657, -0.149658, -0.166305, 0.100652, 0.067567, 0.127259, 0.104348, 0.107074, 0.111429, -0.232715, -0.120531, -0.184443, 0.055374, -0.091313, -0.144675, -0.031590, 0.083564, -0.040816, 0.138746, 0.093717, 0.030608, -0.151200, 0.035843, -0.081479, -0.093672, -0.106533, 0.095600, -0.168453, -0.139404, 0.000521, 0.111324, 0.130851, -0.154690, -0.155250, -0.108958, -0.052336, -0.124921, 0.160949, -0.130016, -0.027504, -0.139416, -0.178927, 0.038461, -0.023239, 0.000045, 0.044404, 0.033308, 0.051093, -0.106325, -0.145973, -0.072122, 0.029732, 0.104050, -0.052619, 0.123613, 0.054704, -0.179320, -0.180839, 0.095339, -0.132829, 0.026997, 0.070502, -0.035763, -0.012464, -0.070170, -0.133024, -0.065789, -0.084381, -0.160771, -0.111578, 0.145180, -0.155922, -0.020064, -0.162391, -0.026823, 0.125361, -0.032008, -0.083072, 0.009838, -0.015261, -0.050777, -0.246227, 0.148361, -0.105394, -0.010375, 0.006983, 0.106619, -0.056164, -0.132590, -0.039194, 0.129358, 0.029220, -0.120276, 0.176940, 0.059489, -0.054668, -0.140159, 0.080929, -0.047651, -0.166564, -0.159694, -0.105646, 0.236992, -0.048422, 0.090006, 0.107739, 0.106466, -0.034345, -0.074629, -0.103216, 0.090364, 0.088547, -0.095429, -0.039066, 0.100523, -0.024857, -0.032562, -0.183530, 0.033953, 0.045317, -0.029822, 0.160822, 0.064885, -0.019779, 0.055399, -0.093930, 0.127363, -0.145180, -0.022765, -0.099703, -0.178664, 0.014401, -0.027952, -0.023255, -0.041077, 0.076452, -0.157341, -0.011823, -0.002641, -0.076511, -0.166012, 0.100003, -0.026833, 0.041142, -0.022881, 0.052015, 0.100347, -0.135295, 0.044829, 0.121359, -0.037871, 0.003639, -0.102953, -0.147525, -0.109356, -0.166415, -0.024267, -0.062384, -0.031624, -0.038623, -0.143746, -0.092854, -0.163245, 0.063375, 0.071740, -0.162606, 0.062290, -0.068545, -0.000434, -0.225524, -0.080865, -0.063993, -0.126933, -0.041284, -0.179465, 0.029988, 0.052810, -0.131245, 0.128665, -0.042853, 0.002494, -0.040490, -0.125760, 0.120420, -0.089038, 0.033506, -0.084146, 0.101011, 0.063219, 0.200410, -0.087390, -0.164569, 0.062727, 0.007944, -0.248787, -0.167678, -0.128019, 0.051793, 0.007865, 0.083040, 0.044476, 0.123940, -0.019675, -0.162633, -0.094126, -0.112904, 0.086950, 0.022722, 0.086028, 0.062676, 0.174804, 0.092907, 0.093094, -0.029311, -0.010211, -0.077123, 0.021141, 0.076186, -0.091854, -0.042958, -0.031239, 0.038252, 0.011443, -0.038989, 0.012473, 0.051853, 0.115186, -0.097301, -0.009709, 0.178788, -0.078586, 0.193954, -0.062569, 0.036496, 0.084922, -0.139171, 0.136011, 0.198799, -0.088511, -0.091240, 0.045427, 0.119364, -0.202744, -0.101552];
    bias_1 : ARRAY[0..95] OF REAL := [0.078665, -0.277721, -0.120379, 0.812712, 0.792883, 0.846731, -0.257424, 0.621971, -0.222661, -0.246470, -0.035770, -0.006102, -0.165188, 0.659960, 0.741415, -0.037438, 0.009055, 0.494007, -0.280266, 0.825763, 0.022478, -0.118515, -0.008948, -0.215567, 0.220641, -0.537282, -0.152418, -0.072453, -0.813448, 0.400618, -0.172556, 0.419335, 0.454605, -0.054706, 0.047425, -0.467890, 0.082506, 0.759780, -0.294553, -0.007059, 0.130478, -0.036144, -0.778336, -0.036332, 0.128106, 0.467416, 0.907125, -0.004070, -0.257575, -0.194332, 0.248056, -0.156112, -0.801525, -0.190145, 0.550399, -0.089834, -0.232022, 0.010967, -0.034462, 0.135814, 0.030903, -0.235148, -0.893473, -0.160944, -0.311711, 0.381273, 0.492836, -0.707353, -1.042032, -0.052282, 0.533243, -0.070562, -0.261179, -0.238909, 0.262229, 0.075838, 0.597456, -0.153160, 0.050517, 0.015945, -0.236519, -0.365638, -0.327759, -0.061266, 0.721874, -0.100470, -0.266727, -0.079038, 0.017814, -1.518959, 0.407458, -0.338946, -0.163797, -0.141941, 0.446652, -0.035327];
